LIN {X 0.105,Y -185.624,Z 1374.736,A 0.000,B 0.000,C 90.000,E1 132.528} C_DIS
LIN {X -0.109,Y -190.219,Z 1374.723,A 0.000,B 0.000,C 90.000,E1 130.092} C_DIS
LIN {X 0.050,Y -197.547,Z 1374.700,A 0.000,B 0.000,C 90.000,E1 125.931} C_DIS
LIN {X -0.069,Y -199.265,Z 1374.695,A 0.000,B 0.000,C 90.000,E1 125.105} C_DIS
LIN {X -0.160,Y -309.469,Z 1374.695,A 0.000,B 0.000,C 90.000,E1 125.105} C_DIS
LIN {X -0.107,Y -315.167,Z 1374.694,A 0.000,B 0.000,C 90.000,E1 124.898} C_DIS
LIN {X 0.002,Y -317.632,Z 1374.693,A 0.000,B 0.000,C 90.000,E1 124.692} C_DIS
LIN {X -0.039,Y -320.942,Z 1374.691,A 0.000,B 0.000,C 90.000,E1 124.326} C_DIS
LIN {X 0.118,Y -322.871,Z 1374.689,A 0.000,B 0.000,C 90.000,E1 123.992} C_DIS
LIN {X 0.008,Y -324.375,Z 1374.687,A 0.000,B 0.000,C 90.000,E1 123.706} C_DIS
LIN {X -0.049,Y -330.062,Z 1374.678,A 0.000,B 0.000,C 90.000,E1 122.133} C_DIS
LIN {X -0.113,Y -341.033,Z 1374.663,A 0.000,B 0.000,C 90.000,E1 119.333} C_DIS
LIN {X -0.049,Y -353.383,Z 1374.648,A 0.000,B 0.000,C 90.000,E1 116.565} C_DIS
LIN {X 0.221,Y -367.224,Z 1374.633,A 0.000,B 0.000,C 90.000,E1 113.823} C_DIS
LIN {X -0.172,Y -380.873,Z 1374.620,A 0.000,B 0.000,C 90.000,E1 111.535} C_DIS
LIN {X -0.009,Y -395.888,Z 1374.607,A 0.000,B 0.000,C 90.000,E1 109.214} C_DIS
LIN {X -0.103,Y -412.375,Z 1374.594,A 0.000,B 0.000,C 90.000,E1 106.985} C_DIS
LIN {X 0.086,Y -430.447,Z 1374.582,A 0.000,B 0.000,C 90.000,E1 104.773} C_DIS
LIN {X 0.229,Y -450.044,Z 1374.570,A 0.000,B 0.000,C 90.000,E1 102.647} C_DIS
LIN {X 0.127,Y -470.327,Z 1374.560,A 0.000,B 0.000,C 90.000,E1 100.715} C_DIS
LIN {X -0.144,Y -483.065,Z 1374.553,A 0.000,B 0.000,C 90.000,E1 99.613} C_DIS
LIN {X -0.024,Y -484.891,Z 1374.552,A 0.000,B 0.000,C 90.000,E1 99.378} C_DIS
LIN {X -0.216,Y -486.450,Z 1374.551,A 0.000,B 0.000,C 90.000,E1 99.151} C_DIS
LIN {X 0.153,Y -487.615,Z 1374.549,A 0.000,B 0.000,C 90.000,E1 98.859} C_DIS
LIN {X -0.131,Y -489.012,Z 1374.547,A 0.000,B 0.000,C 90.000,E1 98.398} C_DIS
LIN {X 0.145,Y -489.364,Z 1374.544,A 0.000,B 0.000,C 90.000,E1 97.871} C_DIS
LIN {X -0.125,Y -488.733,Z 1374.541,A 0.000,B 0.000,C 90.000,E1 97.409} C_DIS
LIN {X 0.092,Y -487.015,Z 1374.538,A 0.000,B 0.000,C 90.000,E1 96.891} C_DIS
LIN {X -0.071,Y -485.649,Z 1374.537,A 0.000,B 0.000,C 90.000,E1 96.663} C_DIS
LIN {X -0.175,Y -473.603,Z 1374.527,A 0.000,B 0.000,C 90.000,E1 94.935} C_DIS
LIN {X 0.126,Y -463.887,Z 1374.519,A 0.000,B 0.000,C 90.000,E1 93.383} C_DIS
LIN {X 0.197,Y -447.231,Z 1374.505,A 0.000,B 0.000,C 90.000,E1 90.802} C_DIS
LIN {X -0.052,Y -430.569,Z 1374.489,A 0.000,B 0.000,C 90.000,E1 87.936} C_DIS
LIN {X 0.031,Y -420.205,Z 1374.478,A 0.000,B 0.000,C 90.000,E1 86.045} C_DIS
LIN {X -0.127,Y -411.195,Z 1374.469,A 0.000,B 0.000,C 90.000,E1 84.432} C_DIS
LIN {X -0.029,Y -402.061,Z 1374.460,A 0.000,B 0.000,C 90.000,E1 82.761} C_DIS
LIN {X -0.049,Y -392.775,Z 1374.450,A 0.000,B 0.000,C 90.000,E1 81.084} C_DIS
LIN {X -0.172,Y -383.322,Z 1374.441,A 0.000,B 0.000,C 90.000,E1 79.398} C_DIS
LIN {X -0.019,Y -373.672,Z 1374.431,A 0.000,B 0.000,C 90.000,E1 77.645} C_DIS
LIN {X 0.006,Y -362.297,Z 1374.420,A 0.000,B 0.000,C 90.000,E1 75.589} C_DIS
LIN {X 0.034,Y -352.345,Z 1374.410,A 0.000,B 0.000,C 90.000,E1 73.795} C_DIS
LIN {X -0.097,Y -340.586,Z 1374.398,A 0.000,B 0.000,C 90.000,E1 71.692} C_DIS
LIN {X -0.079,Y -327.270,Z 1374.384,A 0.000,B 0.000,C 90.000,E1 69.209} C_DIS
LIN {X 0.144,Y -309.803,Z 1374.365,A 0.000,B 0.000,C 90.000,E1 65.665} C_DIS
LIN {X 0.004,Y -298.357,Z 1374.350,A 0.000,B 0.000,C 90.000,E1 63.076} C_DIS
LIN {X -0.008,Y -288.146,Z 1374.336,A 0.000,B 0.000,C 90.000,E1 60.411} C_DIS
LIN {X -0.037,Y -280.120,Z 1374.322,A 0.000,B 0.000,C 90.000,E1 58.043} C_DIS
LIN {X -0.094,Y -269.766,Z 1374.303,A 0.000,B 0.000,C 90.000,E1 54.609} C_DIS
LIN {X 0.025,Y -261.942,Z 1374.288,A 0.000,B 0.000,C 90.000,E1 51.778} C_DIS
LIN {X -0.109,Y -252.668,Z 1374.268,A 0.000,B 0.000,C 90.000,E1 48.243} C_DIS
LIN {X -0.031,Y -243.965,Z 1374.248,A 0.000,B 0.000,C 90.000,E1 44.595} C_DIS
LIN {X -0.046,Y -236.060,Z 1374.227,A 0.000,B 0.000,C 90.000,E1 40.906} C_DIS
LIN {X -0.053,Y -229.071,Z 1374.206,A 0.000,B 0.000,C 90.000,E1 37.156} C_DIS
LIN {X -0.129,Y -223.036,Z 1374.185,A 0.000,B 0.000,C 90.000,E1 33.372} C_DIS
LIN {X -0.004,Y -217.876,Z 1374.164,A 0.000,B 0.000,C 90.000,E1 29.489} C_DIS
LIN {X -0.036,Y -213.025,Z 1374.138,A 0.000,B 0.000,C 90.000,E1 24.823} C_DIS
LIN {X -0.067,Y -209.079,Z 1374.107,A 0.000,B 0.000,C 90.000,E1 19.322} C_DIS
LIN {X -0.103,Y -206.893,Z 1374.085,A 0.000,B 0.000,C 90.000,E1 15.371} C_DIS
LIN {X -0.057,Y -205.266,Z 1374.068,A 0.000,B 0.000,C 90.000,E1 12.175} C_DIS
LIN {X 0.007,Y -203.473,Z 1374.045,A 0.000,B 0.000,C 90.000,E1 8.163} C_DIS
LIN {X 0.081,Y -202.199,Z 1374.028,A 0.000,B 0.000,C 90.000,E1 4.935} C_DIS
LIN {X 0.072,Y -200.811,Z 1374.005,A 0.000,B 0.000,C 90.000,E1 0.917} C_DIS
LIN {X -0.095,Y -199.758,Z 1373.979,A 0.000,B 0.000,C 90.000,E1 356.331} C_DIS
LIN {X -0.074,Y -199.675,Z 1373.944,A 0.000,B 0.000,C 90.000,E1 349.859} C_DIS
LIN {X -0.085,Y -201.962,Z 1373.903,A 0.000,B 0.000,C 90.000,E1 342.598} C_DIS
LIN {X 0.056,Y -205.049,Z 1373.876,A 0.000,B 0.000,C 90.000,E1 337.741} C_DIS
LIN {X 0.008,Y -208.842,Z 1373.854,A 0.000,B 0.000,C 90.000,E1 333.768} C_DIS
LIN {X 0.092,Y -213.731,Z 1373.832,A 0.000,B 0.000,C 90.000,E1 329.793} C_DIS
LIN {X 0.106,Y -219.917,Z 1373.811,A 0.000,B 0.000,C 90.000,E1 325.881} C_DIS
LIN {X -0.049,Y -227.282,Z 1373.789,A 0.000,B 0.000,C 90.000,E1 322.065} C_DIS
LIN {X -0.010,Y -234.219,Z 1373.772,A 0.000,B 0.000,C 90.000,E1 319.013} C_DIS
LIN {X -0.023,Y -242.957,Z 1373.754,A 0.000,B 0.000,C 90.000,E1 315.648} C_DIS
LIN {X -0.114,Y -252.763,Z 1373.735,A 0.000,B 0.000,C 90.000,E1 312.366} C_DIS
LIN {X 0.056,Y -261.458,Z 1373.721,A 0.000,B 0.000,C 90.000,E1 309.806} C_DIS
LIN {X -0.038,Y -272.553,Z 1373.705,A 0.000,B 0.000,C 90.000,E1 306.996} C_DIS
LIN {X 0.034,Y -281.723,Z 1373.694,A 0.000,B 0.000,C 90.000,E1 304.898} C_DIS
LIN {X -0.087,Y -290.252,Z 1373.684,A 0.000,B 0.000,C 90.000,E1 303.214} C_DIS
LIN {X -0.145,Y -299.719,Z 1373.675,A 0.000,B 0.000,C 90.000,E1 301.544} C_DIS
LIN {X -0.081,Y -308.351,Z 1373.668,A 0.000,B 0.000,C 90.000,E1 300.207} C_DIS
LIN {X 0.118,Y -317.891,Z 1373.661,A 0.000,B 0.000,C 90.000,E1 298.871} C_DIS
LIN {X -0.069,Y -341.252,Z 1373.645,A 0.000,B 0.000,C 90.000,E1 296.155} C_DIS
LIN {X 0.073,Y -357.170,Z 1373.635,A 0.000,B 0.000,C 90.000,E1 294.387} C_DIS
LIN {X 0.007,Y -370.314,Z 1373.628,A 0.000,B 0.000,C 90.000,E1 292.950} C_DIS
LIN {X -0.170,Y -383.139,Z 1373.620,A 0.000,B 0.000,C 90.000,E1 291.535} C_DIS
LIN {X 0.068,Y -395.535,Z 1373.612,A 0.000,B 0.000,C 90.000,E1 290.066} C_DIS
LIN {X -0.132,Y -415.163,Z 1373.599,A 0.000,B 0.000,C 90.000,E1 287.873} C_DIS
LIN {X -0.057,Y -422.593,Z 1373.595,A 0.000,B 0.000,C 90.000,E1 287.040} C_DIS
LIN {X 0.097,Y -429.432,Z 1373.590,A 0.000,B 0.000,C 90.000,E1 286.205} C_DIS
LIN {X -0.108,Y -435.752,Z 1373.586,A 0.000,B 0.000,C 90.000,E1 285.426} C_DIS
LIN {X 0.167,Y -441.277,Z 1373.581,A 0.000,B 0.000,C 90.000,E1 284.592} C_DIS
LIN {X -0.050,Y -446.081,Z 1373.577,A 0.000,B 0.000,C 90.000,E1 283.828} C_DIS
LIN {X -0.220,Y -450.004,Z 1373.572,A 0.000,B 0.000,C 90.000,E1 283.063} C_DIS
LIN {X 0.082,Y -453.203,Z 1373.568,A 0.000,B 0.000,C 90.000,E1 282.243} C_DIS
LIN {X 0.156,Y -454.826,Z 1373.565,A 0.000,B 0.000,C 90.000,E1 281.715} C_DIS
LIN {X -0.213,Y -456.108,Z 1373.562,A 0.000,B 0.000,C 90.000,E1 281.243} C_DIS
LIN {X -0.128,Y -456.942,Z 1373.559,A 0.000,B 0.000,C 90.000,E1 280.715} C_DIS
LIN {X -0.118,Y -457.349,Z 1373.557,A 0.000,B 0.000,C 90.000,E1 280.197} C_DIS
LIN {X -0.022,Y -457.353,Z 1373.554,A 0.000,B 0.000,C 90.000,E1 279.670} C_DIS
LIN {X 0.000,Y -456.869,Z 1373.551,A 0.000,B 0.000,C 90.000,E1 279.151} C_DIS
LIN {X 0.094,Y -455.930,Z 1373.548,A 0.000,B 0.000,C 90.000,E1 278.624} C_DIS
LIN {X 0.115,Y -454.459,Z 1373.545,A 0.000,B 0.000,C 90.000,E1 278.106} C_DIS
LIN {X 0.133,Y -452.478,Z 1373.542,A 0.000,B 0.000,C 90.000,E1 277.587} C_DIS
LIN {X 0.144,Y -449.961,Z 1373.539,A 0.000,B 0.000,C 90.000,E1 277.068} C_DIS
LIN {X 0.137,Y -446.826,Z 1373.536,A 0.000,B 0.000,C 90.000,E1 276.549} C_DIS
LIN {X 0.115,Y -442.922,Z 1373.534,A 0.000,B 0.000,C 90.000,E1 276.030} C_DIS
LIN {X 0.072,Y -438.005,Z 1373.531,A 0.000,B 0.000,C 90.000,E1 275.511} C_DIS
LIN {X -0.117,Y -435.182,Z 1373.529,A 0.000,B 0.000,C 90.000,E1 275.277} C_DIS
LIN {X 0.169,Y -429.024,Z 1373.527,A 0.000,B 0.000,C 90.000,E1 274.759} C_DIS
LIN {X 0.043,Y -422.617,Z 1373.524,A 0.000,B 0.000,C 90.000,E1 274.359} C_DIS
LIN {X -0.085,Y -416.040,Z 1373.522,A 0.000,B 0.000,C 90.000,E1 274.012} C_DIS
LIN {X 0.069,Y -409.422,Z 1373.520,A 0.000,B 0.000,C 90.000,E1 273.669} C_DIS
LIN {X -0.047,Y -399.427,Z 1373.518,A 0.000,B 0.000,C 90.000,E1 273.269} C_DIS
LIN {X -0.068,Y -389.737,Z 1373.516,A 0.000,B 0.000,C 90.000,E1 272.922} C_DIS
LIN {X 0.037,Y -382.812,Z 1373.515,A 0.000,B 0.000,C 90.000,E1 272.694} C_DIS
LIN {X -0.053,Y -375.514,Z 1373.514,A 0.000,B 0.000,C 90.000,E1 272.522} C_DIS
LIN {X 0.066,Y -367.884,Z 1373.513,A 0.000,B 0.000,C 90.000,E1 272.350} C_DIS
LIN {X -0.002,Y -356.175,Z 1373.512,A 0.000,B 0.000,C 90.000,E1 272.178} C_DIS
LIN {X 0.066,Y -346.221,Z 1373.511,A 0.000,B 0.000,C 90.000,E1 272.064} C_DIS
LIN {X -0.072,Y -330.914,Z 1373.511,A 0.000,B 0.000,C 90.000,E1 272.007} C_DIS
LIN {X -0.116,Y -327.857,Z 1373.511,A 0.000,B 0.000,C 90.000,E1 272.007} C_DIS
LIN {X -0.089,Y -181.265,Z 1373.511,A 0.000,B 0.000,C 90.000,E1 272.007} C_DIS
LIN {X 0.058,Y -181.581,Z 1373.501,A 0.000,B 0.000,C 90.000,E1 270.229} C_DIS
LIN {X 0.046,Y -180.895,Z 1373.473,A 0.000,B 0.000,C 90.000,E1 265.179} C_DIS
LIN {X 0.053,Y -179.837,Z 1373.459,A 0.000,B 0.000,C 90.000,E1 262.648} C_DIS
LIN {X -0.068,Y -179.024,Z 1373.445,A 0.000,B 0.000,C 90.000,E1 260.151} C_DIS
LIN {X -0.006,Y -178.664,Z 1373.440,A 0.000,B 0.000,C 90.000,E1 259.285} C_DIS
LIN {X -0.070,Y -175.715,Z 1373.412,A 0.000,B 0.000,C 90.000,E1 254.212} C_DIS
LIN {X -0.053,Y -172.430,Z 1373.388,A 0.000,B 0.000,C 90.000,E1 249.934} C_DIS
LIN {X -0.033,Y -171.258,Z 1373.379,A 0.000,B 0.000,C 90.000,E1 248.209} C_DIS
LIN {X -0.050,Y -167.529,Z 1373.355,A 0.000,B 0.000,C 90.000,E1 243.896} C_DIS
LIN {X 0.033,Y -166.925,Z 1373.350,A 0.000,B 0.000,C 90.000,E1 242.999} C_DIS
LIN {X -0.046,Y -162.921,Z 1373.326,A 0.000,B 0.000,C 90.000,E1 238.663} C_DIS
LIN {X -0.068,Y -161.594,Z 1373.316,A 0.000,B 0.000,C 90.000,E1 236.914} C_DIS
LIN {X 0.058,Y -158.336,Z 1373.296,A 0.000,B 0.000,C 90.000,E1 233.336} C_DIS
LIN {X -0.081,Y -155.638,Z 1373.277,A 0.000,B 0.000,C 90.000,E1 229.828} C_DIS
LIN {X -0.026,Y -151.911,Z 1373.252,A 0.000,B 0.000,C 90.000,E1 225.324} C_DIS
LIN {X -0.012,Y -150.145,Z 1373.237,A 0.000,B 0.000,C 90.000,E1 222.609} C_DIS
LIN {X 0.026,Y -146.929,Z 1373.211,A 0.000,B 0.000,C 90.000,E1 218.051} C_DIS
LIN {X 0.017,Y -145.517,Z 1373.196,A 0.000,B 0.000,C 90.000,E1 215.311} C_DIS
LIN {X 0.011,Y -142.917,Z 1373.171,A 0.000,B 0.000,C 90.000,E1 210.718} C_DIS
LIN {X 0.064,Y -141.540,Z 1373.150,A 0.000,B 0.000,C 90.000,E1 207.001} C_DIS
LIN {X -0.024,Y -139.401,Z 1373.114,A 0.000,B 0.000,C 90.000,E1 200.536} C_DIS
LIN {X -0.019,Y -139.118,Z 1373.104,A 0.000,B 0.000,C 90.000,E1 198.671} C_DIS
LIN {X 0.013,Y -138.352,Z 1373.057,A 0.000,B 0.000,C 90.000,E1 190.254} C_DIS
LIN {X 0.003,Y -139.505,Z 1373.005,A 0.000,B 0.000,C 90.000,E1 180.917} C_DIS
LIN {X -0.056,Y -141.138,Z 1372.974,A 0.000,B 0.000,C 90.000,E1 175.355} C_DIS
LIN {X 0.038,Y -142.518,Z 1372.959,A 0.000,B 0.000,C 90.000,E1 172.534} C_DIS
LIN {X -0.017,Y -144.780,Z 1372.933,A 0.000,B 0.000,C 90.000,E1 167.937} C_DIS
LIN {X -0.029,Y -147.396,Z 1372.912,A 0.000,B 0.000,C 90.000,E1 164.267} C_DIS
LIN {X 0.002,Y -149.970,Z 1372.892,A 0.000,B 0.000,C 90.000,E1 160.604} C_DIS
LIN {X 0.012,Y -153.292,Z 1372.872,A 0.000,B 0.000,C 90.000,E1 156.975} C_DIS
LIN {X -0.001,Y -154.996,Z 1372.862,A 0.000,B 0.000,C 90.000,E1 155.177} C_DIS
LIN {X 0.012,Y -158.636,Z 1372.842,A 0.000,B 0.000,C 90.000,E1 151.591} C_DIS
LIN {X -0.051,Y -161.910,Z 1372.827,A 0.000,B 0.000,C 90.000,E1 148.948} C_DIS
LIN {X 0.057,Y -166.100,Z 1372.808,A 0.000,B 0.000,C 90.000,E1 145.388} C_DIS
LIN {X 0.055,Y -171.109,Z 1372.788,A 0.000,B 0.000,C 90.000,E1 141.904} C_DIS
LIN {X -0.026,Y -175.985,Z 1372.769,A 0.000,B 0.000,C 90.000,E1 138.485} C_DIS
LIN {X 0.088,Y -180.232,Z 1372.755,A 0.000,B 0.000,C 90.000,E1 135.891} C_DIS
LIN {X 0.062,Y -185.646,Z 1372.736,A 0.000,B 0.000,C 90.000,E1 132.528} C_DIS
LIN {X 0.115,Y -190.244,Z 1372.723,A 0.000,B 0.000,C 90.000,E1 130.011} C_DIS
LIN {X 0.006,Y -197.572,Z 1372.700,A 0.000,B 0.000,C 90.000,E1 125.931} C_DIS
LIN {X -0.047,Y -199.252,Z 1372.695,A 0.000,B 0.000,C 90.000,E1 125.105} C_DIS
LIN {X -0.125,Y -309.511,Z 1372.695,A 0.000,B 0.000,C 90.000,E1 125.105} C_DIS
LIN {X 0.151,Y -311.252,Z 1372.695,A 0.000,B 0.000,C 90.000,E1 125.025} C_DIS
LIN {X -0.178,Y -315.434,Z 1372.694,A 0.000,B 0.000,C 90.000,E1 124.898} C_DIS
LIN {X -0.069,Y -317.806,Z 1372.693,A 0.000,B 0.000,C 90.000,E1 124.692} C_DIS
LIN {X -0.111,Y -321.038,Z 1372.691,A 0.000,B 0.000,C 90.000,E1 124.326} C_DIS
LIN {X 0.018,Y -322.962,Z 1372.689,A 0.000,B 0.000,C 90.000,E1 123.992} C_DIS
LIN {X -0.122,Y -324.459,Z 1372.687,A 0.000,B 0.000,C 90.000,E1 123.706} C_DIS
LIN {X -0.065,Y -338.549,Z 1372.666,A 0.000,B 0.000,C 90.000,E1 119.922} C_DIS
LIN {X 0.086,Y -350.594,Z 1372.651,A 0.000,B 0.000,C 90.000,E1 117.129} C_DIS
LIN {X -0.208,Y -364.107,Z 1372.636,A 0.000,B 0.000,C 90.000,E1 114.463} C_DIS
LIN {X -0.051,Y -377.441,Z 1372.623,A 0.000,B 0.000,C 90.000,E1 112.078} C_DIS
LIN {X 0.021,Y -392.117,Z 1372.610,A 0.000,B 0.000,C 90.000,E1 109.758} C_DIS
LIN {X -0.043,Y -408.239,Z 1372.597,A 0.000,B 0.000,C 90.000,E1 107.511} C_DIS
LIN {X 0.036,Y -425.918,Z 1372.585,A 0.000,B 0.000,C 90.000,E1 105.300} C_DIS
LIN {X -0.042,Y -445.220,Z 1372.573,A 0.000,B 0.000,C 90.000,E1 103.175} C_DIS
LIN {X -0.025,Y -465.369,Z 1372.562,A 0.000,B 0.000,C 90.000,E1 101.186} C_DIS
LIN {X 0.067,Y -480.831,Z 1372.554,A 0.000,B 0.000,C 90.000,E1 99.792} C_DIS
LIN {X 0.191,Y -483.168,Z 1372.553,A 0.000,B 0.000,C 90.000,E1 99.557} C_DIS
LIN {X -0.165,Y -484.936,Z 1372.552,A 0.000,B 0.000,C 90.000,E1 99.378} C_DIS
LIN {X 0.124,Y -486.450,Z 1372.551,A 0.000,B 0.000,C 90.000,E1 99.095} C_DIS
LIN {X 0.012,Y -487.579,Z 1372.549,A 0.000,B 0.000,C 90.000,E1 98.859} C_DIS
LIN {X 0.212,Y -488.916,Z 1372.547,A 0.000,B 0.000,C 90.000,E1 98.341} C_DIS
LIN {X 0.004,Y -489.218,Z 1372.544,A 0.000,B 0.000,C 90.000,E1 97.871} C_DIS
LIN {X 0.217,Y -488.536,Z 1372.541,A 0.000,B 0.000,C 90.000,E1 97.352} C_DIS
LIN {X -0.050,Y -486.756,Z 1372.538,A 0.000,B 0.000,C 90.000,E1 96.891} C_DIS
LIN {X -0.213,Y -485.350,Z 1372.537,A 0.000,B 0.000,C 90.000,E1 96.663} C_DIS
LIN {X 0.151,Y -473.261,Z 1372.527,A 0.000,B 0.000,C 90.000,E1 94.878} C_DIS
LIN {X -0.022,Y -463.534,Z 1372.519,A 0.000,B 0.000,C 90.000,E1 93.383} C_DIS
LIN {X 0.044,Y -446.887,Z 1372.505,A 0.000,B 0.000,C 90.000,E1 90.802} C_DIS
LIN {X -0.209,Y -430.250,Z 1372.488,A 0.000,B 0.000,C 90.000,E1 87.936} C_DIS
LIN {X -0.129,Y -419.902,Z 1372.478,A 0.000,B 0.000,C 90.000,E1 86.045} C_DIS
LIN {X 0.192,Y -409.407,Z 1372.467,A 0.000,B 0.000,C 90.000,E1 84.090} C_DIS
LIN {X -0.103,Y -400.252,Z 1372.458,A 0.000,B 0.000,C 90.000,E1 82.470} C_DIS
LIN {X -0.150,Y -390.950,Z 1372.449,A 0.000,B 0.000,C 90.000,E1 80.792} C_DIS
LIN {X 0.107,Y -379.869,Z 1372.438,A 0.000,B 0.000,C 90.000,E1 78.757} C_DIS
LIN {X -0.097,Y -368.549,Z 1372.426,A 0.000,B 0.000,C 90.000,E1 76.756} C_DIS
LIN {X -0.132,Y -358.725,Z 1372.417,A 0.000,B 0.000,C 90.000,E1 74.991} C_DIS
LIN {X 0.174,Y -348.741,Z 1372.406,A 0.000,B 0.000,C 90.000,E1 73.142} C_DIS
LIN {X -0.040,Y -336.998,Z 1372.395,A 0.000,B 0.000,C 90.000,E1 71.040} C_DIS
LIN {X -0.008,Y -323.745,Z 1372.381,A 0.000,B 0.000,C 90.000,E1 68.539} C_DIS
LIN {X -0.020,Y -309.564,Z 1372.365,A 0.000,B 0.000,C 90.000,E1 65.665} C_DIS
LIN {X -0.024,Y -298.147,Z 1372.350,A 0.000,B 0.000,C 90.000,E1 63.050} C_DIS
LIN {X -0.040,Y -286.763,Z 1372.334,A 0.000,B 0.000,C 90.000,E1 60.049} C_DIS
LIN {X 0.016,Y -275.761,Z 1372.315,A 0.000,B 0.000,C 90.000,E1 56.628} C_DIS
LIN {X 0.128,Y -265.744,Z 1372.295,A 0.000,B 0.000,C 90.000,E1 53.130} C_DIS
LIN {X -0.020,Y -256.269,Z 1372.276,A 0.000,B 0.000,C 90.000,E1 49.622} C_DIS
LIN {X 0.173,Y -247.360,Z 1372.256,A 0.000,B 0.000,C 90.000,E1 45.972} C_DIS
LIN {X -0.092,Y -239.161,Z 1372.235,A 0.000,B 0.000,C 90.000,E1 42.366} C_DIS
LIN {X -0.033,Y -231.820,Z 1372.214,A 0.000,B 0.000,C 90.000,E1 38.624} C_DIS
LIN {X 0.055,Y -225.418,Z 1372.193,A 0.000,B 0.000,C 90.000,E1 34.818} C_DIS
LIN {X -0.013,Y -219.937,Z 1372.172,A 0.000,B 0.000,C 90.000,E1 31.003} C_DIS
LIN {X -0.017,Y -215.399,Z 1372.151,A 0.000,B 0.000,C 90.000,E1 27.129} C_DIS
LIN {X -0.126,Y -211.288,Z 1372.125,A 0.000,B 0.000,C 90.000,E1 22.461} C_DIS
LIN {X -0.022,Y -208.795,Z 1372.103,A 0.000,B 0.000,C 90.000,E1 18.489} C_DIS
LIN {X -0.064,Y -206.647,Z 1372.081,A 0.000,B 0.000,C 90.000,E1 14.537} C_DIS
LIN {X -0.114,Y -205.032,Z 1372.063,A 0.000,B 0.000,C 90.000,E1 11.366} C_DIS
LIN {X -0.052,Y -203.276,Z 1372.041,A 0.000,B 0.000,C 90.000,E1 7.352} C_DIS
LIN {X -0.003,Y -202.025,Z 1372.023,A 0.000,B 0.000,C 90.000,E1 4.131} C_DIS
LIN {X 0.000,Y -200.675,Z 1372.000,A 0.000,B 0.000,C 90.000,E1 360.000} C_DIS
LIN {X 0.082,Y -199.689,Z 1371.970,A 0.000,B 0.000,C 90.000,E1 354.666} C_DIS
LIN {X -0.016,Y -200.077,Z 1371.935,A 0.000,B 0.000,C 90.000,E1 348.229} C_DIS
LIN {X 0.037,Y -202.542,Z 1371.899,A 0.000,B 0.000,C 90.000,E1 341.764} C_DIS
LIN {X -0.035,Y -205.889,Z 1371.872,A 0.000,B 0.000,C 90.000,E1 336.975} C_DIS
LIN {X -0.051,Y -209.898,Z 1371.850,A 0.000,B 0.000,C 90.000,E1 332.999} C_DIS
LIN {X -0.125,Y -215.041,Z 1371.828,A 0.000,B 0.000,C 90.000,E1 329.076} C_DIS
LIN {X 0.038,Y -221.503,Z 1371.806,A 0.000,B 0.000,C 90.000,E1 325.135} C_DIS
LIN {X 0.003,Y -227.470,Z 1371.789,A 0.000,B 0.000,C 90.000,E1 322.065} C_DIS
LIN {X 0.048,Y -234.398,Z 1371.772,A 0.000,B 0.000,C 90.000,E1 319.013} C_DIS
LIN {X 0.042,Y -243.099,Z 1371.754,A 0.000,B 0.000,C 90.000,E1 315.648} C_DIS
LIN {X -0.042,Y -252.882,Z 1371.735,A 0.000,B 0.000,C 90.000,E1 312.366} C_DIS
LIN {X -0.068,Y -261.572,Z 1371.721,A 0.000,B 0.000,C 90.000,E1 309.850} C_DIS
LIN {X -0.036,Y -271.198,Z 1371.708,A 0.000,B 0.000,C 90.000,E1 307.363} C_DIS
LIN {X 0.121,Y -281.843,Z 1371.694,A 0.000,B 0.000,C 90.000,E1 304.898} C_DIS
LIN {X 0.005,Y -290.386,Z 1371.685,A 0.000,B 0.000,C 90.000,E1 303.214} C_DIS
LIN {X -0.052,Y -297.857,Z 1371.677,A 0.000,B 0.000,C 90.000,E1 301.878} C_DIS
LIN {X -0.027,Y -304.002,Z 1371.672,A 0.000,B 0.000,C 90.000,E1 300.875} C_DIS
LIN {X 0.096,Y -313.091,Z 1371.664,A 0.000,B 0.000,C 90.000,E1 299.539} C_DIS
LIN {X -0.034,Y -323.051,Z 1371.657,A 0.000,B 0.000,C 90.000,E1 298.281} C_DIS
LIN {X -0.070,Y -344.190,Z 1371.644,A 0.000,B 0.000,C 90.000,E1 295.848} C_DIS
LIN {X -0.108,Y -357.584,Z 1371.635,A 0.000,B 0.000,C 90.000,E1 294.387} C_DIS
LIN {X -0.144,Y -370.669,Z 1371.627,A 0.000,B 0.000,C 90.000,E1 292.950} C_DIS
LIN {X 0.171,Y -383.441,Z 1371.619,A 0.000,B 0.000,C 90.000,E1 291.461} C_DIS
LIN {X -0.041,Y -395.776,Z 1371.611,A 0.000,B 0.000,C 90.000,E1 290.066} C_DIS
LIN {X 0.041,Y -415.525,Z 1371.599,A 0.000,B 0.000,C 90.000,E1 287.819} C_DIS
LIN {X 0.122,Y -422.909,Z 1371.594,A 0.000,B 0.000,C 90.000,E1 286.985} C_DIS
LIN {X -0.131,Y -429.736,Z 1371.590,A 0.000,B 0.000,C 90.000,E1 286.205} C_DIS
LIN {X -0.092,Y -434.032,Z 1371.587,A 0.000,B 0.000,C 90.000,E1 285.662} C_DIS
LIN {X 0.160,Y -439.810,Z 1371.583,A 0.000,B 0.000,C 90.000,E1 284.828} C_DIS
LIN {X -0.065,Y -444.862,Z 1371.578,A 0.000,B 0.000,C 90.000,E1 284.064} C_DIS
LIN {X 0.186,Y -449.066,Z 1371.574,A 0.000,B 0.000,C 90.000,E1 283.244} C_DIS
LIN {X 0.046,Y -452.488,Z 1371.569,A 0.000,B 0.000,C 90.000,E1 282.479} C_DIS
LIN {X -0.144,Y -453.489,Z 1371.568,A 0.000,B 0.000,C 90.000,E1 282.243} C_DIS
LIN {X -0.070,Y -455.105,Z 1371.565,A 0.000,B 0.000,C 90.000,E1 281.715} C_DIS
LIN {X 0.010,Y -456.385,Z 1371.562,A 0.000,B 0.000,C 90.000,E1 281.186} C_DIS
LIN {X 0.098,Y -457.229,Z 1371.559,A 0.000,B 0.000,C 90.000,E1 280.658} C_DIS
LIN {X 0.110,Y -457.630,Z 1371.556,A 0.000,B 0.000,C 90.000,E1 280.141} C_DIS
LIN {X 0.208,Y -457.616,Z 1371.554,A 0.000,B 0.000,C 90.000,E1 279.613} C_DIS
LIN {X -0.219,Y -457.147,Z 1371.551,A 0.000,B 0.000,C 90.000,E1 279.151} C_DIS
LIN {X -0.122,Y -456.161,Z 1371.548,A 0.000,B 0.000,C 90.000,E1 278.624} C_DIS
LIN {X -0.099,Y -454.686,Z 1371.545,A 0.000,B 0.000,C 90.000,E1 278.106} C_DIS
LIN {X -0.079,Y -452.731,Z 1371.542,A 0.000,B 0.000,C 90.000,E1 277.587} C_DIS
LIN {X -0.065,Y -450.174,Z 1371.539,A 0.000,B 0.000,C 90.000,E1 277.068} C_DIS
LIN {X -0.069,Y -447.038,Z 1371.536,A 0.000,B 0.000,C 90.000,E1 276.549} C_DIS
LIN {X -0.089,Y -443.104,Z 1371.533,A 0.000,B 0.000,C 90.000,E1 276.030} C_DIS
LIN {X -0.129,Y -438.295,Z 1371.531,A 0.000,B 0.000,C 90.000,E1 275.511} C_DIS
LIN {X -0.126,Y -432.278,Z 1371.528,A 0.000,B 0.000,C 90.000,E1 274.992} C_DIS
LIN {X -0.006,Y -426.017,Z 1371.525,A 0.000,B 0.000,C 90.000,E1 274.531} C_DIS
LIN {X 0.074,Y -419.486,Z 1371.523,A 0.000,B 0.000,C 90.000,E1 274.131} C_DIS
LIN {X 0.181,Y -413.145,Z 1371.521,A 0.000,B 0.000,C 90.000,E1 273.784} C_DIS
LIN {X -0.067,Y -403.447,Z 1371.519,A 0.000,B 0.000,C 90.000,E1 273.383} C_DIS
LIN {X 0.121,Y -393.506,Z 1371.517,A 0.000,B 0.000,C 90.000,E1 272.980} C_DIS
LIN {X -0.149,Y -383.221,Z 1371.515,A 0.000,B 0.000,C 90.000,E1 272.694} C_DIS
LIN {X 0.147,Y -375.886,Z 1371.514,A 0.000,B 0.000,C 90.000,E1 272.465} C_DIS
LIN {X -0.102,Y -368.080,Z 1371.513,A 0.000,B 0.000,C 90.000,E1 272.350} C_DIS
LIN {X -0.126,Y -356.297,Z 1371.512,A 0.000,B 0.000,C 90.000,E1 272.178} C_DIS
LIN {X -0.049,Y -346.546,Z 1371.511,A 0.000,B 0.000,C 90.000,E1 272.064} C_DIS
LIN {X -0.064,Y -336.433,Z 1371.511,A 0.000,B 0.000,C 90.000,E1 272.007} C_DIS
LIN {X 0.108,Y -326.774,Z 1371.511,A 0.000,B 0.000,C 90.000,E1 271.949} C_DIS
LIN {X 0.036,Y -181.268,Z 1371.511,A 0.000,B 0.000,C 90.000,E1 271.949} C_DIS
LIN {X 0.009,Y -181.580,Z 1371.501,A 0.000,B 0.000,C 90.000,E1 270.229} C_DIS
LIN {X -0.002,Y -180.893,Z 1371.473,A 0.000,B 0.000,C 90.000,E1 265.179} C_DIS
LIN {X 0.075,Y -179.517,Z 1371.454,A 0.000,B 0.000,C 90.000,E1 261.781} C_DIS
LIN {X 0.059,Y -179.020,Z 1371.445,A 0.000,B 0.000,C 90.000,E1 260.095} C_DIS
LIN {X -0.055,Y -178.654,Z 1371.440,A 0.000,B 0.000,C 90.000,E1 259.285} C_DIS
LIN {X 0.051,Y -175.705,Z 1371.412,A 0.000,B 0.000,C 90.000,E1 254.157} C_DIS
LIN {X 0.062,Y -172.420,Z 1371.388,A 0.000,B 0.000,C 90.000,E1 249.880} C_DIS
LIN {X 0.078,Y -171.241,Z 1371.379,A 0.000,B 0.000,C 90.000,E1 248.156} C_DIS
LIN {X 0.053,Y -167.518,Z 1371.355,A 0.000,B 0.000,C 90.000,E1 243.845} C_DIS
LIN {X -0.014,Y -166.914,Z 1371.350,A 0.000,B 0.000,C 90.000,E1 242.999} C_DIS
LIN {X 0.038,Y -162.222,Z 1371.321,A 0.000,B 0.000,C 90.000,E1 237.740} C_DIS
LIN {X -0.043,Y -160.803,Z 1371.311,A 0.000,B 0.000,C 90.000,E1 236.008} C_DIS
LIN {X -0.064,Y -157.590,Z 1371.291,A 0.000,B 0.000,C 90.000,E1 232.477} C_DIS
LIN {X -0.006,Y -155.624,Z 1371.277,A 0.000,B 0.000,C 90.000,E1 229.784} C_DIS
LIN {X -0.071,Y -151.901,Z 1371.252,A 0.000,B 0.000,C 90.000,E1 225.324} C_DIS
LIN {X -0.055,Y -150.131,Z 1371.237,A 0.000,B 0.000,C 90.000,E1 222.609} C_DIS
LIN {X 0.073,Y -146.919,Z 1371.211,A 0.000,B 0.000,C 90.000,E1 218.016} C_DIS
LIN {X -0.026,Y -145.507,Z 1371.196,A 0.000,B 0.000,C 90.000,E1 215.311} C_DIS
LIN {X -0.031,Y -142.910,Z 1371.171,A 0.000,B 0.000,C 90.000,E1 210.718} C_DIS
LIN {X 0.022,Y -141.532,Z 1371.150,A 0.000,B 0.000,C 90.000,E1 207.001} C_DIS
LIN {X 0.065,Y -139.398,Z 1371.114,A 0.000,B 0.000,C 90.000,E1 200.482} C_DIS
LIN {X -0.016,Y -139.112,Z 1371.104,A 0.000,B 0.000,C 90.000,E1 198.652} C_DIS
LIN {X -0.029,Y -138.352,Z 1371.057,A 0.000,B 0.000,C 90.000,E1 190.254} C_DIS
LIN {X -0.039,Y -139.507,Z 1371.005,A 0.000,B 0.000,C 90.000,E1 180.917} C_DIS
LIN {X 0.042,Y -141.146,Z 1370.974,A 0.000,B 0.000,C 90.000,E1 175.298} C_DIS
LIN {X -0.006,Y -142.526,Z 1370.958,A 0.000,B 0.000,C 90.000,E1 172.534} C_DIS
LIN {X -0.060,Y -144.791,Z 1370.933,A 0.000,B 0.000,C 90.000,E1 167.937} C_DIS
LIN {X 0.070,Y -147.408,Z 1370.912,A 0.000,B 0.000,C 90.000,E1 164.212} C_DIS
LIN {X -0.042,Y -149.984,Z 1370.892,A 0.000,B 0.000,C 90.000,E1 160.604} C_DIS
LIN {X -0.033,Y -153.309,Z 1370.872,A 0.000,B 0.000,C 90.000,E1 156.975} C_DIS
LIN {X 0.019,Y -155.011,Z 1370.862,A 0.000,B 0.000,C 90.000,E1 155.153} C_DIS
LIN {X 0.042,Y -158.654,Z 1370.842,A 0.000,B 0.000,C 90.000,E1 151.563} C_DIS
LIN {X -0.013,Y -161.931,Z 1370.827,A 0.000,B 0.000,C 90.000,E1 148.918} C_DIS
LIN {X 0.010,Y -166.122,Z 1370.808,A 0.000,B 0.000,C 90.000,E1 145.388} C_DIS
LIN {X 0.007,Y -171.133,Z 1370.788,A 0.000,B 0.000,C 90.000,E1 141.904} C_DIS
LIN {X -0.074,Y -176.009,Z 1370.769,A 0.000,B 0.000,C 90.000,E1 138.485} C_DIS
LIN {X 0.038,Y -180.260,Z 1370.755,A 0.000,B 0.000,C 90.000,E1 135.891} C_DIS
LIN {X 0.012,Y -185.673,Z 1370.736,A 0.000,B 0.000,C 90.000,E1 132.528} C_DIS
LIN {X 0.064,Y -190.274,Z 1370.722,A 0.000,B 0.000,C 90.000,E1 130.011} C_DIS
LIN {X -0.046,Y -197.602,Z 1370.700,A 0.000,B 0.000,C 90.000,E1 125.931} C_DIS
LIN {X -0.030,Y -199.241,Z 1370.695,A 0.000,B 0.000,C 90.000,E1 125.105} C_DIS
LIN {X -0.082,Y -309.283,Z 1370.695,A 0.000,B 0.000,C 90.000,E1 125.105} C_DIS
LIN {X 0.069,Y -311.968,Z 1370.695,A 0.000,B 0.000,C 90.000,E1 125.025} C_DIS
LIN {X 0.179,Y -315.711,Z 1370.694,A 0.000,B 0.000,C 90.000,E1 124.818} C_DIS
LIN {X -0.152,Y -317.990,Z 1370.693,A 0.000,B 0.000,C 90.000,E1 124.692} C_DIS
LIN {X 0.070,Y -321.147,Z 1370.691,A 0.000,B 0.000,C 90.000,E1 124.278} C_DIS
LIN {X -0.097,Y -323.063,Z 1370.689,A 0.000,B 0.000,C 90.000,E1 123.992} C_DIS
LIN {X 0.004,Y -324.552,Z 1370.687,A 0.000,B 0.000,C 90.000,E1 123.658} C_DIS
LIN {X 0.079,Y -338.629,Z 1370.666,A 0.000,B 0.000,C 90.000,E1 119.873} C_DIS
LIN {X -0.065,Y -350.686,Z 1370.651,A 0.000,B 0.000,C 90.000,E1 117.129} C_DIS
LIN {X 0.120,Y -364.213,Z 1370.636,A 0.000,B 0.000,C 90.000,E1 114.387} C_DIS
LIN {X 0.142,Y -377.560,Z 1370.622,A 0.000,B 0.000,C 90.000,E1 112.025} C_DIS
LIN {X -0.139,Y -392.250,Z 1370.610,A 0.000,B 0.000,C 90.000,E1 109.758} C_DIS
LIN {X 0.184,Y -408.386,Z 1370.597,A 0.000,B 0.000,C 90.000,E1 107.457} C_DIS
LIN {X -0.131,Y -426.083,Z 1370.585,A 0.000,B 0.000,C 90.000,E1 105.300} C_DIS
LIN {X 0.223,Y -445.400,Z 1370.573,A 0.000,B 0.000,C 90.000,E1 103.119} C_DIS
LIN {X -0.187,Y -465.554,Z 1370.562,A 0.000,B 0.000,C 90.000,E1 101.186} C_DIS
LIN {X -0.091,Y -481.020,Z 1370.554,A 0.000,B 0.000,C 90.000,E1 99.792} C_DIS
LIN {X 0.034,Y -483.279,Z 1370.553,A 0.000,B 0.000,C 90.000,E1 99.557} C_DIS
LIN {X 0.157,Y -484.988,Z 1370.552,A 0.000,B 0.000,C 90.000,E1 99.321} C_DIS
LIN {X -0.031,Y -486.454,Z 1370.551,A 0.000,B 0.000,C 90.000,E1 99.095} C_DIS
LIN {X -0.145,Y -487.545,Z 1370.549,A 0.000,B 0.000,C 90.000,E1 98.859} C_DIS
LIN {X 0.055,Y -488.821,Z 1370.546,A 0.000,B 0.000,C 90.000,E1 98.341} C_DIS
LIN {X -0.153,Y -489.070,Z 1370.544,A 0.000,B 0.000,C 90.000,E1 97.871} C_DIS
LIN {X 0.060,Y -488.332,Z 1370.541,A 0.000,B 0.000,C 90.000,E1 97.352} C_DIS
LIN {X -0.208,Y -486.485,Z 1370.538,A 0.000,B 0.000,C 90.000,E1 96.891} C_DIS
LIN {X 0.112,Y -485.034,Z 1370.537,A 0.000,B 0.000,C 90.000,E1 96.606} C_DIS
LIN {X -0.008,Y -472.911,Z 1370.527,A 0.000,B 0.000,C 90.000,E1 94.878} C_DIS
LIN {X -0.184,Y -463.183,Z 1370.519,A 0.000,B 0.000,C 90.000,E1 93.383} C_DIS
LIN {X -0.172,Y -443.375,Z 1370.501,A 0.000,B 0.000,C 90.000,E1 90.286} C_DIS
LIN {X 0.195,Y -428.451,Z 1370.487,A 0.000,B 0.000,C 90.000,E1 87.593} C_DIS
LIN {X -0.168,Y -418.087,Z 1370.476,A 0.000,B 0.000,C 90.000,E1 85.755} C_DIS
LIN {X 0.127,Y -407.602,Z 1370.466,A 0.000,B 0.000,C 90.000,E1 83.799} C_DIS
LIN {X 0.150,Y -398.445,Z 1370.456,A 0.000,B 0.000,C 90.000,E1 82.129} C_DIS
LIN {X 0.120,Y -389.103,Z 1370.447,A 0.000,B 0.000,C 90.000,E1 80.443} C_DIS
LIN {X -0.048,Y -378.005,Z 1370.436,A 0.000,B 0.000,C 90.000,E1 78.465} C_DIS
LIN {X 0.077,Y -366.643,Z 1370.425,A 0.000,B 0.000,C 90.000,E1 76.408} C_DIS
LIN {X 0.090,Y -356.793,Z 1370.415,A 0.000,B 0.000,C 90.000,E1 74.629} C_DIS
LIN {X 0.025,Y -346.803,Z 1370.405,A 0.000,B 0.000,C 90.000,E1 72.834} C_DIS
LIN {X 0.091,Y -335.066,Z 1370.393,A 0.000,B 0.000,C 90.000,E1 70.678} C_DIS
LIN {X 0.188,Y -321.857,Z 1370.379,A 0.000,B 0.000,C 90.000,E1 68.156} C_DIS
LIN {X 0.001,Y -307.825,Z 1370.363,A 0.000,B 0.000,C 90.000,E1 65.305} C_DIS
LIN {X 0.081,Y -296.587,Z 1370.348,A 0.000,B 0.000,C 90.000,E1 62.666} C_DIS
LIN {X 0.012,Y -285.419,Z 1370.332,A 0.000,B 0.000,C 90.000,E1 59.665} C_DIS
LIN {X 0.079,Y -275.649,Z 1370.314,A 0.000,B 0.000,C 90.000,E1 56.580} C_DIS
LIN {X -0.036,Y -265.670,Z 1370.295,A 0.000,B 0.000,C 90.000,E1 53.130} C_DIS
LIN {X -0.015,Y -256.223,Z 1370.276,A 0.000,B 0.000,C 90.000,E1 49.585} C_DIS
LIN {X 0.018,Y -247.334,Z 1370.255,A 0.000,B 0.000,C 90.000,E1 45.972} C_DIS
LIN {X 0.094,Y -239.169,Z 1370.235,A 0.000,B 0.000,C 90.000,E1 42.285} C_DIS
LIN {X -0.035,Y -231.863,Z 1370.214,A 0.000,B 0.000,C 90.000,E1 38.588} C_DIS
LIN {X -0.085,Y -225.489,Z 1370.193,A 0.000,B 0.000,C 90.000,E1 34.818} C_DIS
LIN {X -0.147,Y -220.018,Z 1370.172,A 0.000,B 0.000,C 90.000,E1 31.003} C_DIS
LIN {X 0.046,Y -215.517,Z 1370.151,A 0.000,B 0.000,C 90.000,E1 27.078} C_DIS
LIN {X 0.029,Y -211.454,Z 1370.124,A 0.000,B 0.000,C 90.000,E1 22.386} C_DIS
LIN {X -0.071,Y -208.960,Z 1370.103,A 0.000,B 0.000,C 90.000,E1 18.471} C_DIS
LIN {X 0.027,Y -206.795,Z 1370.080,A 0.000,B 0.000,C 90.000,E1 14.481} C_DIS
LIN {X 0.063,Y -204.808,Z 1370.058,A 0.000,B 0.000,C 90.000,E1 10.489} C_DIS
LIN {X 0.082,Y -203.088,Z 1370.036,A 0.000,B 0.000,C 90.000,E1 6.486} C_DIS
LIN {X -0.092,Y -201.556,Z 1370.014,A 0.000,B 0.000,C 90.000,E1 2.522} C_DIS
LIN {X -0.079,Y -200.124,Z 1369.984,A 0.000,B 0.000,C 90.000,E1 357.135} C_DIS
LIN {X -0.098,Y -199.845,Z 1369.948,A 0.000,B 0.000,C 90.000,E1 350.679} C_DIS
LIN {X 0.039,Y -201.876,Z 1369.908,A 0.000,B 0.000,C 90.000,E1 343.378} C_DIS
LIN {X -0.086,Y -205.399,Z 1369.876,A 0.000,B 0.000,C 90.000,E1 337.794} C_DIS
LIN {X 0.067,Y -209.192,Z 1369.854,A 0.000,B 0.000,C 90.000,E1 333.768} C_DIS
LIN {X -0.129,Y -214.111,Z 1369.832,A 0.000,B 0.000,C 90.000,E1 329.871} C_DIS
LIN {X 0.010,Y -220.320,Z 1369.811,A 0.000,B 0.000,C 90.000,E1 325.928} C_DIS
LIN {X 0.053,Y -227.661,Z 1369.789,A 0.000,B 0.000,C 90.000,E1 322.065} C_DIS
LIN {X 0.104,Y -234.575,Z 1369.772,A 0.000,B 0.000,C 90.000,E1 319.013} C_DIS
LIN {X 0.104,Y -243.246,Z 1369.754,A 0.000,B 0.000,C 90.000,E1 315.648} C_DIS
LIN {X 0.027,Y -253.001,Z 1369.735,A 0.000,B 0.000,C 90.000,E1 312.366} C_DIS
LIN {X 0.007,Y -261.679,Z 1369.721,A 0.000,B 0.000,C 90.000,E1 309.850} C_DIS
LIN {X -0.040,Y -272.749,Z 1369.706,A 0.000,B 0.000,C 90.000,E1 307.030} C_DIS
LIN {X -0.025,Y -281.956,Z 1369.694,A 0.000,B 0.000,C 90.000,E1 304.945} C_DIS
LIN {X -0.064,Y -290.515,Z 1369.685,A 0.000,B 0.000,C 90.000,E1 303.245} C_DIS
LIN {X 0.047,Y -299.955,Z 1369.675,A 0.000,B 0.000,C 90.000,E1 301.544} C_DIS
LIN {X 0.089,Y -306.275,Z 1369.670,A 0.000,B 0.000,C 90.000,E1 300.541} C_DIS
LIN {X -0.032,Y -315.592,Z 1369.662,A 0.000,B 0.000,C 90.000,E1 299.255} C_DIS
LIN {X 0.153,Y -328.331,Z 1369.654,A 0.000,B 0.000,C 90.000,E1 297.641} C_DIS
LIN {X -0.103,Y -347.191,Z 1369.642,A 0.000,B 0.000,C 90.000,E1 295.540} C_DIS
LIN {X -0.055,Y -360.443,Z 1369.634,A 0.000,B 0.000,C 90.000,E1 294.079} C_DIS
LIN {X 0.126,Y -370.886,Z 1369.627,A 0.000,B 0.000,C 90.000,E1 292.898} C_DIS
LIN {X 0.058,Y -383.679,Z 1369.619,A 0.000,B 0.000,C 90.000,E1 291.461} C_DIS
LIN {X -0.146,Y -396.016,Z 1369.611,A 0.000,B 0.000,C 90.000,E1 290.066} C_DIS
LIN {X 0.196,Y -413.269,Z 1369.600,A 0.000,B 0.000,C 90.000,E1 288.055} C_DIS
LIN {X -0.012,Y -423.121,Z 1369.594,A 0.000,B 0.000,C 90.000,E1 286.985} C_DIS
LIN {X 0.149,Y -429.947,Z 1369.590,A 0.000,B 0.000,C 90.000,E1 286.150} C_DIS
LIN {X 0.191,Y -434.243,Z 1369.587,A 0.000,B 0.000,C 90.000,E1 285.607} C_DIS
LIN {X 0.026,Y -440.007,Z 1369.582,A 0.000,B 0.000,C 90.000,E1 284.828} C_DIS
LIN {X -0.199,Y -445.048,Z 1369.578,A 0.000,B 0.000,C 90.000,E1 284.064} C_DIS
LIN {X -0.181,Y -447.982,Z 1369.575,A 0.000,B 0.000,C 90.000,E1 283.536} C_DIS
LIN {X 0.103,Y -451.670,Z 1369.571,A 0.000,B 0.000,C 90.000,E1 282.715} C_DIS
LIN {X 0.168,Y -453.700,Z 1369.568,A 0.000,B 0.000,C 90.000,E1 282.187} C_DIS
LIN {X -0.207,Y -455.380,Z 1369.565,A 0.000,B 0.000,C 90.000,E1 281.715} C_DIS
LIN {X -0.126,Y -456.642,Z 1369.562,A 0.000,B 0.000,C 90.000,E1 281.186} C_DIS
LIN {X -0.037,Y -457.484,Z 1369.559,A 0.000,B 0.000,C 90.000,E1 280.658} C_DIS
LIN {X -0.024,Y -457.921,Z 1369.556,A 0.000,B 0.000,C 90.000,E1 280.141} C_DIS
LIN {X 0.077,Y -457.889,Z 1369.553,A 0.000,B 0.000,C 90.000,E1 279.613} C_DIS
LIN {X 0.103,Y -457.420,Z 1369.551,A 0.000,B 0.000,C 90.000,E1 279.095} C_DIS
LIN {X 0.200,Y -456.438,Z 1369.548,A 0.000,B 0.000,C 90.000,E1 278.568} C_DIS
LIN {X -0.226,Y -454.965,Z 1369.545,A 0.000,B 0.000,C 90.000,E1 278.106} C_DIS
LIN {X -0.203,Y -452.973,Z 1369.542,A 0.000,B 0.000,C 90.000,E1 277.587} C_DIS
LIN {X -0.188,Y -450.438,Z 1369.539,A 0.000,B 0.000,C 90.000,E1 277.068} C_DIS
LIN {X -0.139,Y -447.315,Z 1369.536,A 0.000,B 0.000,C 90.000,E1 276.543} C_DIS
LIN {X -0.160,Y -443.449,Z 1369.533,A 0.000,B 0.000,C 90.000,E1 276.024} C_DIS
LIN {X 0.016,Y -441.203,Z 1369.532,A 0.000,B 0.000,C 90.000,E1 275.739} C_DIS
LIN {X 0.009,Y -435.843,Z 1369.529,A 0.000,B 0.000,C 90.000,E1 275.220} C_DIS
LIN {X -0.158,Y -429.767,Z 1369.526,A 0.000,B 0.000,C 90.000,E1 274.759} C_DIS
LIN {X 0.104,Y -423.371,Z 1369.524,A 0.000,B 0.000,C 90.000,E1 274.302} C_DIS
LIN {X -0.026,Y -416.842,Z 1369.522,A 0.000,B 0.000,C 90.000,E1 273.955} C_DIS
LIN {X 0.117,Y -410.309,Z 1369.520,A 0.000,B 0.000,C 90.000,E1 273.612} C_DIS
LIN {X 0.073,Y -403.644,Z 1369.519,A 0.000,B 0.000,C 90.000,E1 273.326} C_DIS
LIN {X -0.180,Y -393.479,Z 1369.516,A 0.000,B 0.000,C 90.000,E1 272.980} C_DIS
LIN {X -0.028,Y -383.338,Z 1369.515,A 0.000,B 0.000,C 90.000,E1 272.636} C_DIS
LIN {X -0.089,Y -375.908,Z 1369.514,A 0.000,B 0.000,C 90.000,E1 272.465} C_DIS
LIN {X 0.067,Y -368.001,Z 1369.513,A 0.000,B 0.000,C 90.000,E1 272.293} C_DIS
LIN {X 0.112,Y -351.817,Z 1369.512,A 0.000,B 0.000,C 90.000,E1 272.064} C_DIS
LIN {X -0.092,Y -340.400,Z 1369.511,A 0.000,B 0.000,C 90.000,E1 272.007} C_DIS
LIN {X 0.065,Y -331.354,Z 1369.511,A 0.000,B 0.000,C 90.000,E1 271.949} C_DIS
LIN {X 0.003,Y -181.270,Z 1369.511,A 0.000,B 0.000,C 90.000,E1 271.949} C_DIS
LIN {X 0.079,Y -181.574,Z 1369.502,A 0.000,B 0.000,C 90.000,E1 270.401} C_DIS
LIN {X 0.040,Y -180.911,Z 1369.476,A 0.000,B 0.000,C 90.000,E1 265.698} C_DIS
LIN {X -0.082,Y -180.827,Z 1369.471,A 0.000,B 0.000,C 90.000,E1 264.894} C_DIS
LIN {X -0.003,Y -178.932,Z 1369.443,A 0.000,B 0.000,C 90.000,E1 259.803} C_DIS
LIN {X 0.036,Y -175.980,Z 1369.415,A 0.000,B 0.000,C 90.000,E1 254.700} C_DIS
LIN {X -0.019,Y -175.472,Z 1369.410,A 0.000,B 0.000,C 90.000,E1 253.866} C_DIS
LIN {X 0.037,Y -172.219,Z 1369.387,A 0.000,B 0.000,C 90.000,E1 249.571} C_DIS
LIN {X 0.016,Y -171.696,Z 1369.382,A 0.000,B 0.000,C 90.000,E1 248.720} C_DIS
LIN {X 0.090,Y -167.290,Z 1369.353,A 0.000,B 0.000,C 90.000,E1 243.512} C_DIS
LIN {X 0.023,Y -166.667,Z 1369.348,A 0.000,B 0.000,C 90.000,E1 242.666} C_DIS
LIN {X -0.062,Y -162.649,Z 1369.324,A 0.000,B 0.000,C 90.000,E1 238.329} C_DIS
LIN {X 0.001,Y -161.338,Z 1369.314,A 0.000,B 0.000,C 90.000,E1 236.548} C_DIS
LIN {X 0.044,Y -157.333,Z 1369.290,A 0.000,B 0.000,C 90.000,E1 232.110} C_DIS
LIN {X -0.023,Y -155.316,Z 1369.275,A 0.000,B 0.000,C 90.000,E1 229.461} C_DIS
LIN {X 0.015,Y -151.671,Z 1369.250,A 0.000,B 0.000,C 90.000,E1 224.960} C_DIS
LIN {X -0.044,Y -150.537,Z 1369.240,A 0.000,B 0.000,C 90.000,E1 223.176} C_DIS
LIN {X -0.011,Y -147.261,Z 1369.215,A 0.000,B 0.000,C 90.000,E1 218.624} C_DIS
LIN {X 0.045,Y -145.288,Z 1369.194,A 0.000,B 0.000,C 90.000,E1 214.945} C_DIS
LIN {X -0.045,Y -142.388,Z 1369.164,A 0.000,B 0.000,C 90.000,E1 209.461} C_DIS
LIN {X 0.001,Y -141.366,Z 1369.148,A 0.000,B 0.000,C 90.000,E1 206.668} C_DIS
LIN {X -0.021,Y -139.344,Z 1369.112,A 0.000,B 0.000,C 90.000,E1 200.174} C_DIS
LIN {X -0.015,Y -139.015,Z 1369.102,A 0.000,B 0.000,C 90.000,E1 198.308} C_DIS
LIN {X -0.019,Y -138.342,Z 1369.055,A 0.000,B 0.000,C 90.000,E1 189.905} C_DIS
LIN {X 0.000,Y -139.395,Z 1369.008,A 0.000,B 0.000,C 90.000,E1 181.489} C_DIS
LIN {X 0.054,Y -141.297,Z 1368.972,A 0.000,B 0.000,C 90.000,E1 174.951} C_DIS
LIN {X 0.011,Y -142.659,Z 1368.957,A 0.000,B 0.000,C 90.000,E1 172.186} C_DIS
LIN {X -0.039,Y -145.002,Z 1368.931,A 0.000,B 0.000,C 90.000,E1 167.589} C_DIS
LIN {X -0.050,Y -147.629,Z 1368.911,A 0.000,B 0.000,C 90.000,E1 163.921} C_DIS
LIN {X 0.029,Y -150.257,Z 1368.890,A 0.000,B 0.000,C 90.000,E1 160.242} C_DIS
LIN {X 0.043,Y -153.655,Z 1368.870,A 0.000,B 0.000,C 90.000,E1 156.613} C_DIS
LIN {X -0.041,Y -157.071,Z 1368.850,A 0.000,B 0.000,C 90.000,E1 153.050} C_DIS
LIN {X 0.038,Y -161.203,Z 1368.830,A 0.000,B 0.000,C 90.000,E1 149.459} C_DIS
LIN {X -0.014,Y -163.295,Z 1368.821,A 0.000,B 0.000,C 90.000,E1 147.709} C_DIS
LIN {X -0.004,Y -167.741,Z 1368.801,A 0.000,B 0.000,C 90.000,E1 144.196} C_DIS
LIN {X -0.092,Y -171.559,Z 1368.787,A 0.000,B 0.000,C 90.000,E1 141.618} C_DIS
LIN {X -0.050,Y -176.503,Z 1368.767,A 0.000,B 0.000,C 90.000,E1 138.162} C_DIS
LIN {X 0.075,Y -180.801,Z 1368.753,A 0.000,B 0.000,C 90.000,E1 135.567} C_DIS
LIN {X 0.060,Y -186.209,Z 1368.735,A 0.000,B 0.000,C 90.000,E1 132.204} C_DIS
LIN {X -0.001,Y -190.846,Z 1368.721,A 0.000,B 0.000,C 90.000,E1 129.725} C_DIS
LIN {X 0.033,Y -196.607,Z 1368.702,A 0.000,B 0.000,C 90.000,E1 126.423} C_DIS
LIN {X 0.004,Y -199.222,Z 1368.695,A 0.000,B 0.000,C 90.000,E1 125.105} C_DIS
LIN {X -0.041,Y -308.952,Z 1368.695,A 0.000,B 0.000,C 90.000,E1 125.105} C_DIS
LIN {X -0.184,Y -310.915,Z 1368.695,A 0.000,B 0.000,C 90.000,E1 125.105} C_DIS
LIN {X -0.086,Y -316.408,Z 1368.693,A 0.000,B 0.000,C 90.000,E1 124.818} C_DIS
LIN {X 0.092,Y -319.535,Z 1368.692,A 0.000,B 0.000,C 90.000,E1 124.485} C_DIS
LIN {X -0.195,Y -323.144,Z 1368.689,A 0.000,B 0.000,C 90.000,E1 123.992} C_DIS
LIN {X 0.065,Y -324.620,Z 1368.687,A 0.000,B 0.000,C 90.000,E1 123.627} C_DIS
LIN {X -0.188,Y -337.441,Z 1368.668,A 0.000,B 0.000,C 90.000,E1 120.207} C_DIS
LIN {X 0.099,Y -349.353,Z 1368.652,A 0.000,B 0.000,C 90.000,E1 117.385} C_DIS
LIN {X -0.077,Y -362.723,Z 1368.637,A 0.000,B 0.000,C 90.000,E1 114.695} C_DIS
LIN {X -0.104,Y -375.921,Z 1368.624,A 0.000,B 0.000,C 90.000,E1 112.333} C_DIS
LIN {X 0.067,Y -390.450,Z 1368.611,A 0.000,B 0.000,C 90.000,E1 109.993} C_DIS
LIN {X -0.167,Y -406.413,Z 1368.599,A 0.000,B 0.000,C 90.000,E1 107.764} C_DIS
LIN {X -0.126,Y -423.921,Z 1368.586,A 0.000,B 0.000,C 90.000,E1 105.552} C_DIS
LIN {X -0.167,Y -443.070,Z 1368.574,A 0.000,B 0.000,C 90.000,E1 103.411} C_DIS
LIN {X 0.153,Y -463.159,Z 1368.563,A 0.000,B 0.000,C 90.000,E1 101.366} C_DIS
LIN {X -0.135,Y -481.165,Z 1368.554,A 0.000,B 0.000,C 90.000,E1 99.782} C_DIS
LIN {X -0.112,Y -483.371,Z 1368.553,A 0.000,B 0.000,C 90.000,E1 99.557} C_DIS
LIN {X -0.204,Y -485.192,Z 1368.552,A 0.000,B 0.000,C 90.000,E1 99.321} C_DIS
LIN {X 0.182,Y -486.563,Z 1368.550,A 0.000,B 0.000,C 90.000,E1 99.029} C_DIS
LIN {X -0.109,Y -488.306,Z 1368.547,A 0.000,B 0.000,C 90.000,E1 98.568} C_DIS
LIN {X 0.091,Y -488.953,Z 1368.545,A 0.000,B 0.000,C 90.000,E1 98.049} C_DIS
LIN {X -0.181,Y -488.615,Z 1368.542,A 0.000,B 0.000,C 90.000,E1 97.587} C_DIS
LIN {X 0.036,Y -487.241,Z 1368.539,A 0.000,B 0.000,C 90.000,E1 97.068} C_DIS
LIN {X -0.069,Y -486.096,Z 1368.538,A 0.000,B 0.000,C 90.000,E1 96.834} C_DIS
LIN {X -0.230,Y -484.563,Z 1368.536,A 0.000,B 0.000,C 90.000,E1 96.606} C_DIS
LIN {X -0.169,Y -474.052,Z 1368.528,A 0.000,B 0.000,C 90.000,E1 95.106} C_DIS
LIN {X -0.071,Y -462.634,Z 1368.518,A 0.000,B 0.000,C 90.000,E1 93.326} C_DIS
LIN {X -0.081,Y -442.889,Z 1368.501,A 0.000,B 0.000,C 90.000,E1 90.229} C_DIS
LIN {X -0.159,Y -427.986,Z 1368.486,A 0.000,B 0.000,C 90.000,E1 87.593} C_DIS
LIN {X 0.179,Y -419.143,Z 1368.478,A 0.000,B 0.000,C 90.000,E1 85.931} C_DIS
LIN {X 0.072,Y -408.666,Z 1368.467,A 0.000,B 0.000,C 90.000,E1 84.033} C_DIS
LIN {X 0.163,Y -399.563,Z 1368.458,A 0.000,B 0.000,C 90.000,E1 82.356} C_DIS
LIN {X 0.095,Y -390.250,Z 1368.448,A 0.000,B 0.000,C 90.000,E1 80.679} C_DIS
LIN {X -0.053,Y -379.165,Z 1368.437,A 0.000,B 0.000,C 90.000,E1 78.701} C_DIS
LIN {X 0.099,Y -369.486,Z 1368.427,A 0.000,B 0.000,C 90.000,E1 76.937} C_DIS
LIN {X 0.072,Y -359.658,Z 1368.418,A 0.000,B 0.000,C 90.000,E1 75.172} C_DIS
LIN {X 0.053,Y -349.722,Z 1368.408,A 0.000,B 0.000,C 90.000,E1 73.378} C_DIS
LIN {X -0.133,Y -337.996,Z 1368.396,A 0.000,B 0.000,C 90.000,E1 71.275} C_DIS
LIN {X -0.067,Y -324.710,Z 1368.382,A 0.000,B 0.000,C 90.000,E1 68.773} C_DIS
LIN {X 0.074,Y -307.440,Z 1368.362,A 0.000,B 0.000,C 90.000,E1 65.229} C_DIS
LIN {X 0.011,Y -296.256,Z 1368.348,A 0.000,B 0.000,C 90.000,E1 62.615} C_DIS
LIN {X -0.048,Y -286.283,Z 1368.333,A 0.000,B 0.000,C 90.000,E1 59.950} C_DIS
LIN {X -0.115,Y -278.523,Z 1368.320,A 0.000,B 0.000,C 90.000,E1 57.582} C_DIS
LIN {X -0.063,Y -268.414,Z 1368.301,A 0.000,B 0.000,C 90.000,E1 54.116} C_DIS
LIN {X -0.024,Y -260.707,Z 1368.285,A 0.000,B 0.000,C 90.000,E1 51.295} C_DIS
LIN {X -0.050,Y -253.373,Z 1368.269,A 0.000,B 0.000,C 90.000,E1 48.447} C_DIS
LIN {X -0.116,Y -244.669,Z 1368.249,A 0.000,B 0.000,C 90.000,E1 44.838} C_DIS
LIN {X -0.104,Y -236.827,Z 1368.229,A 0.000,B 0.000,C 90.000,E1 41.148} C_DIS
LIN {X 0.060,Y -229.840,Z 1368.208,A 0.000,B 0.000,C 90.000,E1 37.363} C_DIS
LIN {X 0.002,Y -223.775,Z 1368.187,A 0.000,B 0.000,C 90.000,E1 33.579} C_DIS
LIN {X -0.042,Y -218.600,Z 1368.165,A 0.000,B 0.000,C 90.000,E1 29.745} C_DIS
LIN {X -0.046,Y -213.753,Z 1368.139,A 0.000,B 0.000,C 90.000,E1 25.079} C_DIS
LIN {X -0.038,Y -209.781,Z 1368.109,A 0.000,B 0.000,C 90.000,E1 19.577} C_DIS
LIN {X 0.011,Y -207.558,Z 1368.087,A 0.000,B 0.000,C 90.000,E1 15.607} C_DIS
LIN {X -0.084,Y -205.493,Z 1368.065,A 0.000,B 0.000,C 90.000,E1 11.658} C_DIS
LIN {X -0.005,Y -203.650,Z 1368.042,A 0.000,B 0.000,C 90.000,E1 7.644} C_DIS
LIN {X 0.074,Y -202.364,Z 1368.025,A 0.000,B 0.000,C 90.000,E1 4.416} C_DIS
LIN {X 0.000,Y -200.857,Z 1368.000,A 0.000,B 0.000,C 90.000,E1 360.000} C_DIS
LIN {X 0.089,Y -199.904,Z 1367.970,A 0.000,B 0.000,C 90.000,E1 354.666} C_DIS
LIN {X 0.003,Y -200.335,Z 1367.935,A 0.000,B 0.000,C 90.000,E1 348.229} C_DIS
LIN {X 0.070,Y -202.866,Z 1367.899,A 0.000,B 0.000,C 90.000,E1 341.764} C_DIS
LIN {X 0.010,Y -206.231,Z 1367.872,A 0.000,B 0.000,C 90.000,E1 336.975} C_DIS
LIN {X 0.006,Y -210.243,Z 1367.850,A 0.000,B 0.000,C 90.000,E1 332.999} C_DIS
LIN {X -0.054,Y -215.431,Z 1367.828,A 0.000,B 0.000,C 90.000,E1 329.076} C_DIS
LIN {X -0.059,Y -221.892,Z 1367.807,A 0.000,B 0.000,C 90.000,E1 325.182} C_DIS
LIN {X -0.079,Y -227.840,Z 1367.789,A 0.000,B 0.000,C 90.000,E1 322.110} C_DIS
LIN {X -0.020,Y -234.735,Z 1367.772,A 0.000,B 0.000,C 90.000,E1 319.057} C_DIS
LIN {X -0.005,Y -243.392,Z 1367.754,A 0.000,B 0.000,C 90.000,E1 315.688} C_DIS
LIN {X 0.093,Y -253.123,Z 1367.735,A 0.000,B 0.000,C 90.000,E1 312.366} C_DIS
LIN {X 0.078,Y -261.788,Z 1367.721,A 0.000,B 0.000,C 90.000,E1 309.850} C_DIS
LIN {X 0.122,Y -271.415,Z 1367.708,A 0.000,B 0.000,C 90.000,E1 307.363} C_DIS
LIN {X 0.058,Y -282.067,Z 1367.694,A 0.000,B 0.000,C 90.000,E1 304.945} C_DIS
LIN {X 0.164,Y -292.430,Z 1367.683,A 0.000,B 0.000,C 90.000,E1 302.880} C_DIS
LIN {X -0.114,Y -302.086,Z 1367.674,A 0.000,B 0.000,C 90.000,E1 301.258} C_DIS
LIN {X -0.022,Y -310.924,Z 1367.666,A 0.000,B 0.000,C 90.000,E1 299.922} C_DIS
LIN {X 0.158,Y -320.501,Z 1367.659,A 0.000,B 0.000,C 90.000,E1 298.615} C_DIS
LIN {X 0.035,Y -344.355,Z 1367.644,A 0.000,B 0.000,C 90.000,E1 295.848} C_DIS
LIN {X 0.052,Y -357.616,Z 1367.635,A 0.000,B 0.000,C 90.000,E1 294.387} C_DIS
LIN {X -0.018,Y -370.737,Z 1367.627,A 0.000,B 0.000,C 90.000,E1 292.950} C_DIS
LIN {X 0.115,Y -383.514,Z 1367.619,A 0.000,B 0.000,C 90.000,E1 291.482} C_DIS
LIN {X -0.010,Y -395.952,Z 1367.611,A 0.000,B 0.000,C 90.000,E1 290.066} C_DIS
LIN {X -0.056,Y -413.170,Z 1367.601,A 0.000,B 0.000,C 90.000,E1 288.109} C_DIS
LIN {X -0.222,Y -422.937,Z 1367.594,A 0.000,B 0.000,C 90.000,E1 287.040} C_DIS
LIN {X -0.067,Y -429.800,Z 1367.590,A 0.000,B 0.000,C 90.000,E1 286.205} C_DIS
LIN {X 0.148,Y -436.103,Z 1367.585,A 0.000,B 0.000,C 90.000,E1 285.371} C_DIS
LIN {X 0.005,Y -441.715,Z 1367.581,A 0.000,B 0.000,C 90.000,E1 284.592} C_DIS
LIN {X -0.210,Y -446.514,Z 1367.577,A 0.000,B 0.000,C 90.000,E1 283.828} C_DIS
LIN {X -0.182,Y -449.279,Z 1367.574,A 0.000,B 0.000,C 90.000,E1 283.300} C_DIS
LIN {X -0.134,Y -451.699,Z 1367.571,A 0.000,B 0.000,C 90.000,E1 282.771} C_DIS
LIN {X -0.072,Y -453.769,Z 1367.568,A 0.000,B 0.000,C 90.000,E1 282.243} C_DIS
LIN {X 0.005,Y -455.474,Z 1367.565,A 0.000,B 0.000,C 90.000,E1 281.715} C_DIS
LIN {X 0.086,Y -456.816,Z 1367.562,A 0.000,B 0.000,C 90.000,E1 281.186} C_DIS
LIN {X 0.177,Y -457.675,Z 1367.559,A 0.000,B 0.000,C 90.000,E1 280.658} C_DIS
LIN {X 0.192,Y -458.182,Z 1367.557,A 0.000,B 0.000,C 90.000,E1 280.141} C_DIS
LIN {X -0.159,Y -458.230,Z 1367.554,A 0.000,B 0.000,C 90.000,E1 279.670} C_DIS
LIN {X -0.132,Y -457.773,Z 1367.551,A 0.000,B 0.000,C 90.000,E1 279.151} C_DIS
LIN {X -0.033,Y -456.844,Z 1367.548,A 0.000,B 0.000,C 90.000,E1 278.624} C_DIS
LIN {X -0.005,Y -455.410,Z 1367.545,A 0.000,B 0.000,C 90.000,E1 278.106} C_DIS
LIN {X 0.019,Y -453.452,Z 1367.542,A 0.000,B 0.000,C 90.000,E1 277.587} C_DIS
LIN {X 0.035,Y -450.964,Z 1367.539,A 0.000,B 0.000,C 90.000,E1 277.068} C_DIS
LIN {X 0.035,Y -447.890,Z 1367.536,A 0.000,B 0.000,C 90.000,E1 276.549} C_DIS
LIN {X 0.019,Y -444.128,Z 1367.534,A 0.000,B 0.000,C 90.000,E1 276.030} C_DIS
LIN {X -0.016,Y -439.473,Z 1367.531,A 0.000,B 0.000,C 90.000,E1 275.511} C_DIS
LIN {X 0.191,Y -436.741,Z 1367.529,A 0.000,B 0.000,C 90.000,E1 275.220} C_DIS
LIN {X -0.076,Y -433.641,Z 1367.528,A 0.000,B 0.000,C 90.000,E1 274.992} C_DIS
LIN {X -0.039,Y -427.377,Z 1367.525,A 0.000,B 0.000,C 90.000,E1 274.531} C_DIS
LIN {X -0.030,Y -420.900,Z 1367.523,A 0.000,B 0.000,C 90.000,E1 274.131} C_DIS
LIN {X -0.026,Y -414.388,Z 1367.521,A 0.000,B 0.000,C 90.000,E1 273.784} C_DIS
LIN {X 0.091,Y -404.831,Z 1367.519,A 0.000,B 0.000,C 90.000,E1 273.326} C_DIS
LIN {X -0.186,Y -394.723,Z 1367.516,A 0.000,B 0.000,C 90.000,E1 272.980} C_DIS
LIN {X -0.042,Y -384.714,Z 1367.515,A 0.000,B 0.000,C 90.000,E1 272.636} C_DIS
LIN {X -0.103,Y -377.518,Z 1367.514,A 0.000,B 0.000,C 90.000,E1 272.465} C_DIS
LIN {X 0.025,Y -369.624,Z 1367.513,A 0.000,B 0.000,C 90.000,E1 272.293} C_DIS
LIN {X 0.095,Y -353.607,Z 1367.512,A 0.000,B 0.000,C 90.000,E1 272.064} C_DIS
LIN {X -0.113,Y -343.664,Z 1367.511,A 0.000,B 0.000,C 90.000,E1 272.007} C_DIS
LIN {X -0.071,Y -329.797,Z 1367.511,A 0.000,B 0.000,C 90.000,E1 271.949} C_DIS
LIN {X -0.062,Y -181.274,Z 1367.511,A 0.000,B 0.000,C 90.000,E1 271.949} C_DIS
LIN {X -0.090,Y -181.580,Z 1367.501,A 0.000,B 0.000,C 90.000,E1 270.229} C_DIS
LIN {X 0.080,Y -180.889,Z 1367.473,A 0.000,B 0.000,C 90.000,E1 265.122} C_DIS
LIN {X -0.037,Y -179.013,Z 1367.445,A 0.000,B 0.000,C 90.000,E1 260.095} C_DIS
LIN {X 0.057,Y -178.633,Z 1367.440,A 0.000,B 0.000,C 90.000,E1 259.218} C_DIS
LIN {X -0.045,Y -175.684,Z 1367.412,A 0.000,B 0.000,C 90.000,E1 254.157} C_DIS
LIN {X -0.034,Y -172.401,Z 1367.388,A 0.000,B 0.000,C 90.000,E1 249.880} C_DIS
LIN {X -0.017,Y -171.210,Z 1367.379,A 0.000,B 0.000,C 90.000,E1 248.156} C_DIS
LIN {X 0.033,Y -167.495,Z 1367.355,A 0.000,B 0.000,C 90.000,E1 243.819} C_DIS
LIN {X 0.041,Y -166.892,Z 1367.350,A 0.000,B 0.000,C 90.000,E1 242.948} C_DIS
LIN {X 0.032,Y -162.197,Z 1367.321,A 0.000,B 0.000,C 90.000,E1 237.709} C_DIS
LIN {X -0.001,Y -160.770,Z 1367.311,A 0.000,B 0.000,C 90.000,E1 235.960} C_DIS
LIN {X -0.029,Y -157.565,Z 1367.291,A 0.000,B 0.000,C 90.000,E1 232.431} C_DIS
LIN {X 0.005,Y -155.596,Z 1367.276,A 0.000,B 0.000,C 90.000,E1 229.747} C_DIS
LIN {X 0.056,Y -151.877,Z 1367.251,A 0.000,B 0.000,C 90.000,E1 225.243} C_DIS
LIN {X 0.069,Y -150.103,Z 1367.236,A 0.000,B 0.000,C 90.000,E1 222.528} C_DIS
LIN {X -0.014,Y -146.899,Z 1367.211,A 0.000,B 0.000,C 90.000,E1 218.016} C_DIS
LIN {X 0.006,Y -145.487,Z 1367.196,A 0.000,B 0.000,C 90.000,E1 215.264} C_DIS
LIN {X 0.006,Y -142.895,Z 1367.170,A 0.000,B 0.000,C 90.000,E1 210.669} C_DIS
LIN {X -0.063,Y -141.515,Z 1367.150,A 0.000,B 0.000,C 90.000,E1 207.001} C_DIS
LIN {X -0.019,Y -139.393,Z 1367.114,A 0.000,B 0.000,C 90.000,E1 200.482} C_DIS
LIN {X 0.032,Y -139.103,Z 1367.103,A 0.000,B 0.000,C 90.000,E1 198.598} C_DIS
LIN {X 0.024,Y -138.354,Z 1367.057,A 0.000,B 0.000,C 90.000,E1 190.197} C_DIS
LIN {X 0.017,Y -139.513,Z 1367.005,A 0.000,B 0.000,C 90.000,E1 180.859} C_DIS
LIN {X -0.043,Y -141.161,Z 1366.974,A 0.000,B 0.000,C 90.000,E1 175.298} C_DIS
LIN {X 0.069,Y -142.540,Z 1366.958,A 0.000,B 0.000,C 90.000,E1 172.470} C_DIS
LIN {X -0.004,Y -144.812,Z 1366.933,A 0.000,B 0.000,C 90.000,E1 167.881} C_DIS
LIN {X -0.017,Y -147.431,Z 1366.912,A 0.000,B 0.000,C 90.000,E1 164.212} C_DIS
LIN {X 0.012,Y -150.010,Z 1366.892,A 0.000,B 0.000,C 90.000,E1 160.550} C_DIS
LIN {X 0.019,Y -153.343,Z 1366.872,A 0.000,B 0.000,C 90.000,E1 156.922} C_DIS
LIN {X 0.000,Y -155.878,Z 1366.857,A 0.000,B 0.000,C 90.000,E1 154.229} C_DIS
LIN {X -0.034,Y -159.733,Z 1366.837,A 0.000,B 0.000,C 90.000,E1 150.667} C_DIS
LIN {X 0.032,Y -161.972,Z 1366.827,A 0.000,B 0.000,C 90.000,E1 148.869} C_DIS
LIN {X -0.083,Y -166.164,Z 1366.807,A 0.000,B 0.000,C 90.000,E1 145.388} C_DIS
LIN {X -0.089,Y -171.177,Z 1366.788,A 0.000,B 0.000,C 90.000,E1 141.904} C_DIS
LIN {X 0.077,Y -176.059,Z 1366.769,A 0.000,B 0.000,C 90.000,E1 138.405} C_DIS
LIN {X -0.059,Y -180.315,Z 1366.755,A 0.000,B 0.000,C 90.000,E1 135.891} C_DIS
LIN {X -0.088,Y -185.726,Z 1366.736,A 0.000,B 0.000,C 90.000,E1 132.528} C_DIS
LIN {X -0.037,Y -190.334,Z 1366.722,A 0.000,B 0.000,C 90.000,E1 130.011} C_DIS
LIN {X 0.011,Y -197.660,Z 1366.699,A 0.000,B 0.000,C 90.000,E1 125.884} C_DIS
LIN {X 0.022,Y -199.212,Z 1366.695,A 0.000,B 0.000,C 90.000,E1 125.105} C_DIS
LIN {X -0.018,Y -309.156,Z 1366.695,A 0.000,B 0.000,C 90.000,E1 125.105} C_DIS
LIN {X -0.174,Y -311.045,Z 1366.695,A 0.000,B 0.000,C 90.000,E1 125.105} C_DIS
LIN {X -0.026,Y -314.380,Z 1366.694,A 0.000,B 0.000,C 90.000,E1 124.945} C_DIS
LIN {X 0.006,Y -317.732,Z 1366.693,A 0.000,B 0.000,C 90.000,E1 124.692} C_DIS
LIN {X 0.049,Y -321.389,Z 1366.690,A 0.000,B 0.000,C 90.000,E1 124.246} C_DIS
LIN {X 0.133,Y -323.244,Z 1366.688,A 0.000,B 0.000,C 90.000,E1 123.913} C_DIS
LIN {X -0.051,Y -324.686,Z 1366.687,A 0.000,B 0.000,C 90.000,E1 123.627} C_DIS
LIN {X 0.166,Y -337.493,Z 1366.667,A 0.000,B 0.000,C 90.000,E1 120.129} C_DIS
LIN {X -0.014,Y -349.418,Z 1366.652,A 0.000,B 0.000,C 90.000,E1 117.385} C_DIS
LIN {X 0.141,Y -362.793,Z 1366.637,A 0.000,B 0.000,C 90.000,E1 114.643} C_DIS
LIN {X 0.131,Y -376.000,Z 1366.624,A 0.000,B 0.000,C 90.000,E1 112.280} C_DIS
LIN {X -0.049,Y -390.538,Z 1366.611,A 0.000,B 0.000,C 90.000,E1 109.993} C_DIS
LIN {X 0.227,Y -406.512,Z 1366.599,A 0.000,B 0.000,C 90.000,E1 107.692} C_DIS
LIN {X -0.133,Y -424.031,Z 1366.586,A 0.000,B 0.000,C 90.000,E1 105.536} C_DIS
LIN {X 0.144,Y -443.188,Z 1366.574,A 0.000,B 0.000,C 90.000,E1 103.355} C_DIS
LIN {X 0.037,Y -463.280,Z 1366.563,A 0.000,B 0.000,C 90.000,E1 101.366} C_DIS
LIN {X 0.208,Y -481.308,Z 1366.554,A 0.000,B 0.000,C 90.000,E1 99.726} C_DIS
LIN {X -0.253,Y -483.451,Z 1366.553,A 0.000,B 0.000,C 90.000,E1 99.557} C_DIS
LIN {X -0.159,Y -485.079,Z 1366.552,A 0.000,B 0.000,C 90.000,E1 99.321} C_DIS
LIN {X 0.209,Y -486.454,Z 1366.550,A 0.000,B 0.000,C 90.000,E1 99.029} C_DIS
LIN {X 0.020,Y -487.471,Z 1366.549,A 0.000,B 0.000,C 90.000,E1 98.803} C_DIS
LIN {X -0.191,Y -488.626,Z 1366.546,A 0.000,B 0.000,C 90.000,E1 98.333} C_DIS
LIN {X 0.013,Y -488.767,Z 1366.543,A 0.000,B 0.000,C 90.000,E1 97.814} C_DIS
LIN {X 0.225,Y -487.917,Z 1366.541,A 0.000,B 0.000,C 90.000,E1 97.296} C_DIS
LIN {X -0.044,Y -485.932,Z 1366.538,A 0.000,B 0.000,C 90.000,E1 96.834} C_DIS
LIN {X -0.208,Y -484.387,Z 1366.537,A 0.000,B 0.000,C 90.000,E1 96.606} C_DIS
LIN {X -0.149,Y -473.850,Z 1366.528,A 0.000,B 0.000,C 90.000,E1 95.106} C_DIS
LIN {X 0.154,Y -464.052,Z 1366.520,A 0.000,B 0.000,C 90.000,E1 93.555} C_DIS
LIN {X 0.043,Y -452.320,Z 1366.510,A 0.000,B 0.000,C 90.000,E1 91.776} C_DIS
LIN {X 0.035,Y -438.116,Z 1366.497,A 0.000,B 0.000,C 90.000,E1 89.427} C_DIS
LIN {X -0.019,Y -426.320,Z 1366.485,A 0.000,B 0.000,C 90.000,E1 87.306} C_DIS
LIN {X -0.104,Y -417.463,Z 1366.476,A 0.000,B 0.000,C 90.000,E1 85.698} C_DIS
LIN {X 0.175,Y -406.999,Z 1366.465,A 0.000,B 0.000,C 90.000,E1 83.742} C_DIS
LIN {X -0.208,Y -397.882,Z 1366.456,A 0.000,B 0.000,C 90.000,E1 82.129} C_DIS
LIN {X 0.142,Y -388.536,Z 1366.447,A 0.000,B 0.000,C 90.000,E1 80.387} C_DIS
LIN {X -0.040,Y -377.448,Z 1366.436,A 0.000,B 0.000,C 90.000,E1 78.409} C_DIS
LIN {X 0.079,Y -367.718,Z 1366.426,A 0.000,B 0.000,C 90.000,E1 76.645} C_DIS
LIN {X 0.071,Y -356.227,Z 1366.414,A 0.000,B 0.000,C 90.000,E1 74.574} C_DIS
LIN {X -0.006,Y -346.258,Z 1366.404,A 0.000,B 0.000,C 90.000,E1 72.779} C_DIS
LIN {X 0.156,Y -334.531,Z 1366.392,A 0.000,B 0.000,C 90.000,E1 70.604} C_DIS
LIN {X 0.126,Y -321.336,Z 1366.378,A 0.000,B 0.000,C 90.000,E1 68.103} C_DIS
LIN {X -0.044,Y -305.859,Z 1366.361,A 0.000,B 0.000,C 90.000,E1 64.921} C_DIS
LIN {X -0.006,Y -294.868,Z 1366.346,A 0.000,B 0.000,C 90.000,E1 62.281} C_DIS
LIN {X 0.046,Y -285.039,Z 1366.331,A 0.000,B 0.000,C 90.000,E1 59.587} C_DIS
LIN {X 0.152,Y -273.338,Z 1366.310,A 0.000,B 0.000,C 90.000,E1 55.801} C_DIS
LIN {X -0.012,Y -265.492,Z 1366.295,A 0.000,B 0.000,C 90.000,E1 53.050} C_DIS
LIN {X 0.006,Y -256.115,Z 1366.275,A 0.000,B 0.000,C 90.000,E1 49.504} C_DIS
LIN {X 0.036,Y -247.289,Z 1366.255,A 0.000,B 0.000,C 90.000,E1 45.891} C_DIS
LIN {X -0.051,Y -239.183,Z 1366.235,A 0.000,B 0.000,C 90.000,E1 42.243} C_DIS
LIN {X -0.020,Y -231.951,Z 1366.214,A 0.000,B 0.000,C 90.000,E1 38.508} C_DIS
LIN {X -0.071,Y -225.616,Z 1366.193,A 0.000,B 0.000,C 90.000,E1 34.739} C_DIS
LIN {X 0.055,Y -220.175,Z 1366.172,A 0.000,B 0.000,C 90.000,E1 30.875} C_DIS
LIN {X 0.059,Y -215.745,Z 1366.150,A 0.000,B 0.000,C 90.000,E1 27.001} C_DIS
LIN {X -0.038,Y -211.748,Z 1366.124,A 0.000,B 0.000,C 90.000,E1 22.333} C_DIS
LIN {X 0.034,Y -208.810,Z 1366.098,A 0.000,B 0.000,C 90.000,E1 17.583} C_DIS
LIN {X -0.012,Y -207.069,Z 1366.080,A 0.000,B 0.000,C 90.000,E1 14.426} C_DIS
LIN {X 0.036,Y -205.048,Z 1366.058,A 0.000,B 0.000,C 90.000,E1 10.433} C_DIS
LIN {X 0.064,Y -203.257,Z 1366.036,A 0.000,B 0.000,C 90.000,E1 6.429} C_DIS
LIN {X 0.098,Y -201.701,Z 1366.014,A 0.000,B 0.000,C 90.000,E1 2.407} C_DIS
LIN {X -0.076,Y -200.303,Z 1365.984,A 0.000,B 0.000,C 90.000,E1 357.135} C_DIS
LIN {X -0.085,Y -200.072,Z 1365.948,A 0.000,B 0.000,C 90.000,E1 350.679} C_DIS
LIN {X 0.065,Y -202.169,Z 1365.908,A 0.000,B 0.000,C 90.000,E1 343.378} C_DIS
LIN {X -0.046,Y -205.729,Z 1365.877,A 0.000,B 0.000,C 90.000,E1 337.794} C_DIS
LIN {X -0.069,Y -209.536,Z 1365.854,A 0.000,B 0.000,C 90.000,E1 333.819} C_DIS
LIN {X -0.065,Y -214.495,Z 1365.833,A 0.000,B 0.000,C 90.000,E1 329.871} C_DIS
LIN {X -0.035,Y -220.691,Z 1365.811,A 0.000,B 0.000,C 90.000,E1 325.960} C_DIS
LIN {X -0.034,Y -228.021,Z 1365.789,A 0.000,B 0.000,C 90.000,E1 322.110} C_DIS
LIN {X 0.032,Y -234.893,Z 1365.773,A 0.000,B 0.000,C 90.000,E1 319.057} C_DIS
LIN {X -0.121,Y -243.541,Z 1365.754,A 0.000,B 0.000,C 90.000,E1 315.729} C_DIS
LIN {X -0.023,Y -252.098,Z 1365.738,A 0.000,B 0.000,C 90.000,E1 312.771} C_DIS
LIN {X -0.065,Y -260.608,Z 1365.724,A 0.000,B 0.000,C 90.000,E1 310.253} C_DIS
LIN {X 0.124,Y -270.095,Z 1365.710,A 0.000,B 0.000,C 90.000,E1 307.729} C_DIS
LIN {X 0.029,Y -280.586,Z 1365.696,A 0.000,B 0.000,C 90.000,E1 305.311} C_DIS
LIN {X 0.136,Y -288.969,Z 1365.687,A 0.000,B 0.000,C 90.000,E1 303.579} C_DIS
LIN {X -0.033,Y -298.208,Z 1365.677,A 0.000,B 0.000,C 90.000,E1 301.926} C_DIS
LIN {X -0.007,Y -304.308,Z 1365.672,A 0.000,B 0.000,C 90.000,E1 300.924} C_DIS
LIN {X -0.038,Y -313.343,Z 1365.665,A 0.000,B 0.000,C 90.000,E1 299.617} C_DIS
LIN {X -0.069,Y -325.842,Z 1365.656,A 0.000,B 0.000,C 90.000,E1 298.025} C_DIS
LIN {X -0.066,Y -346.970,Z 1365.642,A 0.000,B 0.000,C 90.000,E1 295.591} C_DIS
LIN {X -0.104,Y -360.275,Z 1365.634,A 0.000,B 0.000,C 90.000,E1 294.131} C_DIS
LIN {X 0.148,Y -370.639,Z 1365.628,A 0.000,B 0.000,C 90.000,E1 292.950} C_DIS
LIN {X -0.041,Y -383.347,Z 1365.620,A 0.000,B 0.000,C 90.000,E1 291.535} C_DIS
LIN {X -0.177,Y -395.787,Z 1365.612,A 0.000,B 0.000,C 90.000,E1 290.120} C_DIS
LIN {X 0.026,Y -412.970,Z 1365.601,A 0.000,B 0.000,C 90.000,E1 288.127} C_DIS
LIN {X -0.041,Y -422.767,Z 1365.595,A 0.000,B 0.000,C 90.000,E1 287.040} C_DIS
LIN {X -0.139,Y -431.852,Z 1365.589,A 0.000,B 0.000,C 90.000,E1 285.969} C_DIS
LIN {X 0.102,Y -437.946,Z 1365.584,A 0.000,B 0.000,C 90.000,E1 285.134} C_DIS
LIN {X 0.189,Y -441.639,Z 1365.581,A 0.000,B 0.000,C 90.000,E1 284.592} C_DIS
LIN {X -0.025,Y -446.510,Z 1365.577,A 0.000,B 0.000,C 90.000,E1 283.828} C_DIS
LIN {X 0.004,Y -449.303,Z 1365.574,A 0.000,B 0.000,C 90.000,E1 283.300} C_DIS
LIN {X -0.136,Y -452.864,Z 1365.570,A 0.000,B 0.000,C 90.000,E1 282.535} C_DIS
LIN {X 0.194,Y -455.568,Z 1365.565,A 0.000,B 0.000,C 90.000,E1 281.715} C_DIS
LIN {X -0.171,Y -456.962,Z 1365.562,A 0.000,B 0.000,C 90.000,E1 281.243} C_DIS
LIN {X -0.081,Y -457.896,Z 1365.559,A 0.000,B 0.000,C 90.000,E1 280.715} C_DIS
LIN {X -0.067,Y -458.443,Z 1365.557,A 0.000,B 0.000,C 90.000,E1 280.197} C_DIS
LIN {X 0.035,Y -458.514,Z 1365.554,A 0.000,B 0.000,C 90.000,E1 279.670} C_DIS
LIN {X 0.063,Y -458.104,Z 1365.551,A 0.000,B 0.000,C 90.000,E1 279.151} C_DIS
LIN {X 0.165,Y -457.237,Z 1365.548,A 0.000,B 0.000,C 90.000,E1 278.624} C_DIS
LIN {X 0.193,Y -455.826,Z 1365.545,A 0.000,B 0.000,C 90.000,E1 278.106} C_DIS
LIN {X -0.232,Y -453.941,Z 1365.542,A 0.000,B 0.000,C 90.000,E1 277.644} C_DIS
LIN {X -0.212,Y -451.466,Z 1365.539,A 0.000,B 0.000,C 90.000,E1 277.125} C_DIS
LIN {X -0.208,Y -448.451,Z 1365.536,A 0.000,B 0.000,C 90.000,E1 276.606} C_DIS
LIN {X -0.220,Y -444.784,Z 1365.534,A 0.000,B 0.000,C 90.000,E1 276.087} C_DIS
LIN {X 0.189,Y -440.280,Z 1365.531,A 0.000,B 0.000,C 90.000,E1 275.511} C_DIS
LIN {X 0.131,Y -434.581,Z 1365.528,A 0.000,B 0.000,C 90.000,E1 274.992} C_DIS
LIN {X 0.094,Y -428.406,Z 1365.525,A 0.000,B 0.000,C 90.000,E1 274.531} C_DIS
LIN {X 0.049,Y -421.933,Z 1365.523,A 0.000,B 0.000,C 90.000,E1 274.131} C_DIS
LIN {X 0.111,Y -412.300,Z 1365.520,A 0.000,B 0.000,C 90.000,E1 273.612} C_DIS
LIN {X 0.038,Y -405.740,Z 1365.519,A 0.000,B 0.000,C 90.000,E1 273.326} C_DIS
LIN {X 0.138,Y -395.703,Z 1365.516,A 0.000,B 0.000,C 90.000,E1 272.922} C_DIS
LIN {X -0.167,Y -385.396,Z 1365.515,A 0.000,B 0.000,C 90.000,E1 272.636} C_DIS
LIN {X 0.102,Y -378.050,Z 1365.513,A 0.000,B 0.000,C 90.000,E1 272.407} C_DIS
LIN {X -0.158,Y -369.783,Z 1365.513,A 0.000,B 0.000,C 90.000,E1 272.293} C_DIS
LIN {X -0.069,Y -353.418,Z 1365.511,A 0.000,B 0.000,C 90.000,E1 272.064} C_DIS
LIN {X 0.075,Y -343.366,Z 1365.511,A 0.000,B 0.000,C 90.000,E1 271.949} C_DIS
LIN {X 0.154,Y -330.440,Z 1365.511,A 0.000,B 0.000,C 90.000,E1 271.892} C_DIS
LIN {X 0.065,Y -181.276,Z 1365.511,A 0.000,B 0.000,C 90.000,E1 271.892} C_DIS
LIN {X 0.045,Y -181.579,Z 1365.501,A 0.000,B 0.000,C 90.000,E1 270.172} C_DIS
LIN {X 0.033,Y -180.887,Z 1365.473,A 0.000,B 0.000,C 90.000,E1 265.122} C_DIS
LIN {X -0.084,Y -179.009,Z 1365.445,A 0.000,B 0.000,C 90.000,E1 260.095} C_DIS
LIN {X 0.010,Y -178.622,Z 1365.440,A 0.000,B 0.000,C 90.000,E1 259.218} C_DIS
LIN {X 0.078,Y -175.674,Z 1365.412,A 0.000,B 0.000,C 90.000,E1 254.102} C_DIS
LIN {X -0.079,Y -172.391,Z 1365.388,A 0.000,B 0.000,C 90.000,E1 249.880} C_DIS
LIN {X -0.062,Y -171.195,Z 1365.379,A 0.000,B 0.000,C 90.000,E1 248.156} C_DIS
LIN {X -0.011,Y -167.484,Z 1365.354,A 0.000,B 0.000,C 90.000,E1 243.819} C_DIS
LIN {X -0.003,Y -166.881,Z 1365.350,A 0.000,B 0.000,C 90.000,E1 242.948} C_DIS
LIN {X -0.011,Y -162.186,Z 1365.321,A 0.000,B 0.000,C 90.000,E1 237.709} C_DIS
LIN {X 0.046,Y -160.755,Z 1365.311,A 0.000,B 0.000,C 90.000,E1 235.928} C_DIS
LIN {X 0.025,Y -157.552,Z 1365.291,A 0.000,B 0.000,C 90.000,E1 232.396} C_DIS
LIN {X -0.037,Y -155.581,Z 1365.276,A 0.000,B 0.000,C 90.000,E1 229.747} C_DIS
LIN {X 0.014,Y -151.866,Z 1365.251,A 0.000,B 0.000,C 90.000,E1 225.243} C_DIS
LIN {X 0.028,Y -150.090,Z 1365.236,A 0.000,B 0.000,C 90.000,E1 222.528} C_DIS
LIN {X -0.054,Y -146.891,Z 1365.211,A 0.000,B 0.000,C 90.000,E1 218.016} C_DIS
LIN {X 0.050,Y -145.477,Z 1365.196,A 0.000,B 0.000,C 90.000,E1 215.231} C_DIS
LIN {X -0.033,Y -142.888,Z 1365.170,A 0.000,B 0.000,C 90.000,E1 210.669} C_DIS
LIN {X 0.024,Y -141.507,Z 1365.150,A 0.000,B 0.000,C 90.000,E1 206.950} C_DIS
LIN {X -0.059,Y -139.391,Z 1365.114,A 0.000,B 0.000,C 90.000,E1 200.482} C_DIS
LIN {X -0.007,Y -139.098,Z 1365.103,A 0.000,B 0.000,C 90.000,E1 198.598} C_DIS
LIN {X -0.016,Y -138.354,Z 1365.057,A 0.000,B 0.000,C 90.000,E1 190.197} C_DIS
LIN {X -0.023,Y -139.515,Z 1365.005,A 0.000,B 0.000,C 90.000,E1 180.859} C_DIS
LIN {X 0.058,Y -141.168,Z 1364.974,A 0.000,B 0.000,C 90.000,E1 175.241} C_DIS
LIN {X 0.029,Y -142.547,Z 1364.958,A 0.000,B 0.000,C 90.000,E1 172.470} C_DIS
LIN {X -0.045,Y -144.822,Z 1364.933,A 0.000,B 0.000,C 90.000,E1 167.881} C_DIS
LIN {X -0.058,Y -147.443,Z 1364.912,A 0.000,B 0.000,C 90.000,E1 164.212} C_DIS
LIN {X -0.030,Y -150.024,Z 1364.892,A 0.000,B 0.000,C 90.000,E1 160.550} C_DIS
LIN {X -0.024,Y -153.360,Z 1364.872,A 0.000,B 0.000,C 90.000,E1 156.922} C_DIS
LIN {X 0.025,Y -155.893,Z 1364.857,A 0.000,B 0.000,C 90.000,E1 154.204} C_DIS
LIN {X -0.077,Y -159.751,Z 1364.837,A 0.000,B 0.000,C 90.000,E1 150.667} C_DIS
LIN {X -0.011,Y -161.991,Z 1364.827,A 0.000,B 0.000,C 90.000,E1 148.869} C_DIS
LIN {X 0.009,Y -166.184,Z 1364.807,A 0.000,B 0.000,C 90.000,E1 145.341} C_DIS
LIN {X 0.107,Y -171.199,Z 1364.788,A 0.000,B 0.000,C 90.000,E1 141.823} C_DIS
LIN {X 0.031,Y -176.081,Z 1364.769,A 0.000,B 0.000,C 90.000,E1 138.405} C_DIS
LIN {X -0.107,Y -180.342,Z 1364.755,A 0.000,B 0.000,C 90.000,E1 135.891} C_DIS
LIN {X 0.001,Y -185.752,Z 1364.736,A 0.000,B 0.000,C 90.000,E1 132.486} C_DIS
LIN {X -0.085,Y -190.363,Z 1364.722,A 0.000,B 0.000,C 90.000,E1 130.011} C_DIS
LIN {X -0.039,Y -197.689,Z 1364.699,A 0.000,B 0.000,C 90.000,E1 125.884} C_DIS
LIN {X 0.025,Y -199.209,Z 1364.695,A 0.000,B 0.000,C 90.000,E1 125.105} C_DIS
LIN {X 0.004,Y -309.141,Z 1364.695,A 0.000,B 0.000,C 90.000,E1 125.105} C_DIS
LIN {X 0.182,Y -311.691,Z 1364.695,A 0.000,B 0.000,C 90.000,E1 125.025} C_DIS
LIN {X 0.094,Y -314.849,Z 1364.694,A 0.000,B 0.000,C 90.000,E1 124.898} C_DIS
LIN {X 0.121,Y -318.345,Z 1364.692,A 0.000,B 0.000,C 90.000,E1 124.612} C_DIS
LIN {X -0.201,Y -321.966,Z 1364.690,A 0.000,B 0.000,C 90.000,E1 124.199} C_DIS
LIN {X 0.054,Y -323.690,Z 1364.688,A 0.000,B 0.000,C 90.000,E1 123.833} C_DIS
LIN {X -0.048,Y -326.132,Z 1364.684,A 0.000,B 0.000,C 90.000,E1 123.214} C_DIS
LIN {X -0.056,Y -336.603,Z 1364.669,A 0.000,B 0.000,C 90.000,E1 120.384} C_DIS
LIN {X 0.039,Y -348.414,Z 1364.653,A 0.000,B 0.000,C 90.000,E1 117.590} C_DIS
LIN {X -0.158,Y -361.676,Z 1364.638,A 0.000,B 0.000,C 90.000,E1 114.899} C_DIS
LIN {X -0.061,Y -374.771,Z 1364.625,A 0.000,B 0.000,C 90.000,E1 112.514} C_DIS
LIN {X 0.078,Y -389.190,Z 1364.612,A 0.000,B 0.000,C 90.000,E1 110.174} C_DIS
LIN {X -0.186,Y -405.034,Z 1364.600,A 0.000,B 0.000,C 90.000,E1 107.946} C_DIS
LIN {X -0.066,Y -422.413,Z 1364.587,A 0.000,B 0.000,C 90.000,E1 105.717} C_DIS
LIN {X 0.153,Y -441.448,Z 1364.575,A 0.000,B 0.000,C 90.000,E1 103.536} C_DIS
LIN {X 0.023,Y -461.490,Z 1364.564,A 0.000,B 0.000,C 90.000,E1 101.535} C_DIS
LIN {X 0.116,Y -481.976,Z 1364.554,A 0.000,B 0.000,C 90.000,E1 99.670} C_DIS
LIN {X 0.094,Y -483.954,Z 1364.552,A 0.000,B 0.000,C 90.000,E1 99.443} C_DIS
LIN {X 0.153,Y -485.461,Z 1364.551,A 0.000,B 0.000,C 90.000,E1 99.208} C_DIS
LIN {X 0.042,Y -486.704,Z 1364.550,A 0.000,B 0.000,C 90.000,E1 98.973} C_DIS
LIN {X -0.145,Y -487.612,Z 1364.548,A 0.000,B 0.000,C 90.000,E1 98.746} C_DIS
LIN {X 0.129,Y -488.585,Z 1364.546,A 0.000,B 0.000,C 90.000,E1 98.219} C_DIS
LIN {X -0.149,Y -488.558,Z 1364.543,A 0.000,B 0.000,C 90.000,E1 97.757} C_DIS
LIN {X 0.065,Y -487.530,Z 1364.540,A 0.000,B 0.000,C 90.000,E1 97.239} C_DIS
LIN {X -0.041,Y -486.593,Z 1364.539,A 0.000,B 0.000,C 90.000,E1 97.004} C_DIS
LIN {X -0.205,Y -485.319,Z 1364.537,A 0.000,B 0.000,C 90.000,E1 96.777} C_DIS
LIN {X 0.004,Y -471.489,Z 1364.526,A 0.000,B 0.000,C 90.000,E1 94.759} C_DIS
LIN {X -0.233,Y -461.610,Z 1364.518,A 0.000,B 0.000,C 90.000,E1 93.269} C_DIS
LIN {X -0.084,Y -440.425,Z 1364.499,A 0.000,B 0.000,C 90.000,E1 89.885} C_DIS
LIN {X 0.061,Y -427.112,Z 1364.486,A 0.000,B 0.000,C 90.000,E1 87.478} C_DIS
LIN {X -0.010,Y -418.286,Z 1364.477,A 0.000,B 0.000,C 90.000,E1 85.869} C_DIS
LIN {X -0.057,Y -406.339,Z 1364.465,A 0.000,B 0.000,C 90.000,E1 83.685} C_DIS
LIN {X 0.001,Y -397.215,Z 1364.456,A 0.000,B 0.000,C 90.000,E1 82.008} C_DIS
LIN {X -0.105,Y -387.880,Z 1364.446,A 0.000,B 0.000,C 90.000,E1 80.330} C_DIS
LIN {X 0.149,Y -376.790,Z 1364.435,A 0.000,B 0.000,C 90.000,E1 78.285} C_DIS
LIN {X -0.185,Y -367.068,Z 1364.425,A 0.000,B 0.000,C 90.000,E1 76.589} C_DIS
LIN {X -0.201,Y -355.568,Z 1364.414,A 0.000,B 0.000,C 90.000,E1 74.519} C_DIS
LIN {X 0.044,Y -345.582,Z 1364.404,A 0.000,B 0.000,C 90.000,E1 72.670} C_DIS
LIN {X -0.142,Y -332.207,Z 1364.390,A 0.000,B 0.000,C 90.000,E1 70.242} C_DIS
LIN {X 0.138,Y -317.496,Z 1364.374,A 0.000,B 0.000,C 90.000,E1 67.358} C_DIS
LIN {X 0.088,Y -303.838,Z 1364.358,A 0.000,B 0.000,C 90.000,E1 64.460} C_DIS
LIN {X 0.074,Y -294.356,Z 1364.345,A 0.000,B 0.000,C 90.000,E1 62.153} C_DIS
LIN {X 0.135,Y -285.726,Z 1364.332,A 0.000,B 0.000,C 90.000,E1 59.793} C_DIS
LIN {X -0.130,Y -277.050,Z 1364.317,A 0.000,B 0.000,C 90.000,E1 57.120} C_DIS
LIN {X 0.025,Y -267.110,Z 1364.298,A 0.000,B 0.000,C 90.000,E1 53.623} C_DIS
LIN {X -0.072,Y -257.662,Z 1364.278,A 0.000,B 0.000,C 90.000,E1 50.114} C_DIS
LIN {X 0.011,Y -248.758,Z 1364.258,A 0.000,B 0.000,C 90.000,E1 46.500} C_DIS
LIN {X -0.032,Y -240.530,Z 1364.238,A 0.000,B 0.000,C 90.000,E1 42.852} C_DIS
LIN {X 0.042,Y -233.214,Z 1364.217,A 0.000,B 0.000,C 90.000,E1 39.116} C_DIS
LIN {X -0.017,Y -226.715,Z 1364.196,A 0.000,B 0.000,C 90.000,E1 35.358} C_DIS
LIN {X -0.047,Y -221.137,Z 1364.175,A 0.000,B 0.000,C 90.000,E1 31.544} C_DIS
LIN {X 0.093,Y -216.544,Z 1364.154,A 0.000,B 0.000,C 90.000,E1 27.641} C_DIS
LIN {X 0.109,Y -212.378,Z 1364.128,A 0.000,B 0.000,C 90.000,E1 22.950} C_DIS
LIN {X 0.072,Y -209.336,Z 1364.101,A 0.000,B 0.000,C 90.000,E1 18.236} C_DIS
LIN {X -0.017,Y -207.110,Z 1364.079,A 0.000,B 0.000,C 90.000,E1 14.300} C_DIS
LIN {X 0.024,Y -205.089,Z 1364.057,A 0.000,B 0.000,C 90.000,E1 10.310} C_DIS
LIN {X 0.020,Y -203.288,Z 1364.035,A 0.000,B 0.000,C 90.000,E1 6.315} C_DIS
LIN {X 0.057,Y -201.724,Z 1364.013,A 0.000,B 0.000,C 90.000,E1 2.293} C_DIS
LIN {X -0.084,Y -200.248,Z 1363.979,A 0.000,B 0.000,C 90.000,E1 356.331} C_DIS
LIN {X -0.037,Y -200.268,Z 1363.944,A 0.000,B 0.000,C 90.000,E1 349.859} C_DIS
LIN {X -0.010,Y -202.714,Z 1363.903,A 0.000,B 0.000,C 90.000,E1 342.598} C_DIS
LIN {X -0.028,Y -205.892,Z 1363.877,A 0.000,B 0.000,C 90.000,E1 337.794} C_DIS
LIN {X -0.046,Y -209.705,Z 1363.854,A 0.000,B 0.000,C 90.000,E1 333.819} C_DIS
LIN {X -0.036,Y -214.676,Z 1363.833,A 0.000,B 0.000,C 90.000,E1 329.871} C_DIS
LIN {X 0.001,Y -220.874,Z 1363.811,A 0.000,B 0.000,C 90.000,E1 325.960} C_DIS
LIN {X 0.009,Y -228.196,Z 1363.790,A 0.000,B 0.000,C 90.000,E1 322.110} C_DIS
LIN {X -0.074,Y -235.051,Z 1363.773,A 0.000,B 0.000,C 90.000,E1 319.094} C_DIS
LIN {X -0.066,Y -243.690,Z 1363.754,A 0.000,B 0.000,C 90.000,E1 315.729} C_DIS
LIN {X 0.038,Y -252.225,Z 1363.738,A 0.000,B 0.000,C 90.000,E1 312.771} C_DIS
LIN {X 0.001,Y -260.730,Z 1363.724,A 0.000,B 0.000,C 90.000,E1 310.253} C_DIS
LIN {X -0.184,Y -270.221,Z 1363.710,A 0.000,B 0.000,C 90.000,E1 307.810} C_DIS
LIN {X 0.105,Y -280.701,Z 1363.696,A 0.000,B 0.000,C 90.000,E1 305.311} C_DIS
LIN {X -0.024,Y -289.075,Z 1363.687,A 0.000,B 0.000,C 90.000,E1 303.627} C_DIS
LIN {X 0.052,Y -298.320,Z 1363.677,A 0.000,B 0.000,C 90.000,E1 301.926} C_DIS
LIN {X 0.100,Y -306.602,Z 1363.670,A 0.000,B 0.000,C 90.000,E1 300.590} C_DIS
LIN {X 0.102,Y -315.847,Z 1363.663,A 0.000,B 0.000,C 90.000,E1 299.283} C_DIS
LIN {X 0.001,Y -333.890,Z 1363.650,A 0.000,B 0.000,C 90.000,E1 297.078} C_DIS
LIN {X -0.056,Y -349.886,Z 1363.640,A 0.000,B 0.000,C 90.000,E1 295.283} C_DIS
LIN {X -0.083,Y -363.171,Z 1363.632,A 0.000,B 0.000,C 90.000,E1 293.823} C_DIS
LIN {X -0.016,Y -370.980,Z 1363.627,A 0.000,B 0.000,C 90.000,E1 292.950} C_DIS
LIN {X 0.111,Y -383.717,Z 1363.619,A 0.000,B 0.000,C 90.000,E1 291.482} C_DIS
LIN {X -0.005,Y -396.128,Z 1363.611,A 0.000,B 0.000,C 90.000,E1 290.066} C_DIS
LIN {X 0.127,Y -410.801,Z 1363.602,A 0.000,B 0.000,C 90.000,E1 288.362} C_DIS
LIN {X 0.014,Y -420.685,Z 1363.596,A 0.000,B 0.000,C 90.000,E1 287.275} C_DIS
LIN {X 0.142,Y -427.697,Z 1363.591,A 0.000,B 0.000,C 90.000,E1 286.441} C_DIS
LIN {X -0.071,Y -434.235,Z 1363.587,A 0.000,B 0.000,C 90.000,E1 285.662} C_DIS
LIN {X 0.184,Y -440.121,Z 1363.583,A 0.000,B 0.000,C 90.000,E1 284.828} C_DIS
LIN {X -0.038,Y -445.252,Z 1363.578,A 0.000,B 0.000,C 90.000,E1 284.064} C_DIS
LIN {X -0.017,Y -448.255,Z 1363.575,A 0.000,B 0.000,C 90.000,E1 283.536} C_DIS
LIN {X -0.172,Y -452.026,Z 1363.571,A 0.000,B 0.000,C 90.000,E1 282.771} C_DIS
LIN {X -0.107,Y -454.109,Z 1363.568,A 0.000,B 0.000,C 90.000,E1 282.243} C_DIS
LIN {X -0.029,Y -455.817,Z 1363.565,A 0.000,B 0.000,C 90.000,E1 281.715} C_DIS
LIN {X 0.055,Y -457.187,Z 1363.562,A 0.000,B 0.000,C 90.000,E1 281.186} C_DIS
LIN {X 0.147,Y -458.192,Z 1363.559,A 0.000,B 0.000,C 90.000,E1 280.658} C_DIS
LIN {X 0.164,Y -458.709,Z 1363.556,A 0.000,B 0.000,C 90.000,E1 280.141} C_DIS
LIN {X -0.184,Y -458.813,Z 1363.554,A 0.000,B 0.000,C 90.000,E1 279.670} C_DIS
LIN {X -0.154,Y -458.394,Z 1363.551,A 0.000,B 0.000,C 90.000,E1 279.151} C_DIS
LIN {X -0.051,Y -457.508,Z 1363.548,A 0.000,B 0.000,C 90.000,E1 278.624} C_DIS
LIN {X -0.020,Y -456.135,Z 1363.545,A 0.000,B 0.000,C 90.000,E1 278.106} C_DIS
LIN {X 0.007,Y -454.221,Z 1363.542,A 0.000,B 0.000,C 90.000,E1 277.587} C_DIS
LIN {X 0.028,Y -451.727,Z 1363.539,A 0.000,B 0.000,C 90.000,E1 277.068} C_DIS
LIN {X 0.033,Y -448.663,Z 1363.536,A 0.000,B 0.000,C 90.000,E1 276.549} C_DIS
LIN {X 0.022,Y -445.021,Z 1363.534,A 0.000,B 0.000,C 90.000,E1 276.030} C_DIS
LIN {X -0.009,Y -440.552,Z 1363.531,A 0.000,B 0.000,C 90.000,E1 275.511} C_DIS
LIN {X -0.063,Y -434.887,Z 1363.528,A 0.000,B 0.000,C 90.000,E1 274.992} C_DIS
LIN {X -0.116,Y -428.733,Z 1363.525,A 0.000,B 0.000,C 90.000,E1 274.531} C_DIS
LIN {X -0.102,Y -422.419,Z 1363.523,A 0.000,B 0.000,C 90.000,E1 274.131} C_DIS
LIN {X -0.169,Y -415.922,Z 1363.521,A 0.000,B 0.000,C 90.000,E1 273.784} C_DIS
LIN {X -0.195,Y -406.087,Z 1363.518,A 0.000,B 0.000,C 90.000,E1 273.326} C_DIS
LIN {X -0.119,Y -395.928,Z 1363.516,A 0.000,B 0.000,C 90.000,E1 272.922} C_DIS
LIN {X -0.007,Y -385.743,Z 1363.514,A 0.000,B 0.000,C 90.000,E1 272.579} C_DIS
LIN {X -0.098,Y -378.430,Z 1363.513,A 0.000,B 0.000,C 90.000,E1 272.407} C_DIS
LIN {X 0.029,Y -370.167,Z 1363.512,A 0.000,B 0.000,C 90.000,E1 272.236} C_DIS
LIN {X -0.148,Y -349.311,Z 1363.511,A 0.000,B 0.000,C 90.000,E1 272.007} C_DIS
LIN {X 0.086,Y -335.143,Z 1363.511,A 0.000,B 0.000,C 90.000,E1 271.892} C_DIS
LIN {X 0.013,Y -181.279,Z 1363.510,A 0.000,B 0.000,C 90.000,E1 271.892} C_DIS
LIN {X 0.088,Y -181.578,Z 1363.502,A 0.000,B 0.000,C 90.000,E1 270.344} C_DIS
LIN {X -0.075,Y -180.809,Z 1363.471,A 0.000,B 0.000,C 90.000,E1 264.837} C_DIS
LIN {X 0.002,Y -178.911,Z 1363.443,A 0.000,B 0.000,C 90.000,E1 259.746} C_DIS
LIN {X 0.082,Y -175.955,Z 1363.415,A 0.000,B 0.000,C 90.000,E1 254.629} C_DIS
LIN {X 0.028,Y -175.424,Z 1363.410,A 0.000,B 0.000,C 90.000,E1 253.795} C_DIS
LIN {X 0.030,Y -172.185,Z 1363.386,A 0.000,B 0.000,C 90.000,E1 249.518} C_DIS
LIN {X 0.070,Y -171.656,Z 1363.381,A 0.000,B 0.000,C 90.000,E1 248.646} C_DIS
LIN {X 0.064,Y -167.881,Z 1363.358,A 0.000,B 0.000,C 90.000,E1 244.332} C_DIS
LIN {X 0.007,Y -166.617,Z 1363.348,A 0.000,B 0.000,C 90.000,E1 242.615} C_DIS
LIN {X 0.000,Y -162.605,Z 1363.324,A 0.000,B 0.000,C 90.000,E1 238.250} C_DIS
LIN {X -0.025,Y -161.289,Z 1363.314,A 0.000,B 0.000,C 90.000,E1 236.501} C_DIS
LIN {X 0.009,Y -157.288,Z 1363.289,A 0.000,B 0.000,C 90.000,E1 232.065} C_DIS
LIN {X 0.032,Y -156.006,Z 1363.279,A 0.000,B 0.000,C 90.000,E1 230.275} C_DIS
LIN {X -0.008,Y -152.264,Z 1363.255,A 0.000,B 0.000,C 90.000,E1 225.810} C_DIS
LIN {X 0.014,Y -150.501,Z 1363.240,A 0.000,B 0.000,C 90.000,E1 223.095} C_DIS
LIN {X 0.044,Y -147.226,Z 1363.214,A 0.000,B 0.000,C 90.000,E1 218.543} C_DIS
LIN {X 0.013,Y -145.248,Z 1363.194,A 0.000,B 0.000,C 90.000,E1 214.898} C_DIS
LIN {X -0.070,Y -142.365,Z 1363.163,A 0.000,B 0.000,C 90.000,E1 209.411} C_DIS
LIN {X 0.051,Y -141.751,Z 1363.153,A 0.000,B 0.000,C 90.000,E1 207.513} C_DIS
LIN {X -0.024,Y -139.494,Z 1363.117,A 0.000,B 0.000,C 90.000,E1 201.046} C_DIS
LIN {X 0.013,Y -138.998,Z 1363.101,A 0.000,B 0.000,C 90.000,E1 198.236} C_DIS
LIN {X -0.030,Y -138.337,Z 1363.055,A 0.000,B 0.000,C 90.000,E1 189.849} C_DIS
LIN {X -0.008,Y -139.411,Z 1363.008,A 0.000,B 0.000,C 90.000,E1 181.432} C_DIS
LIN {X 0.045,Y -141.324,Z 1362.972,A 0.000,B 0.000,C 90.000,E1 174.894} C_DIS
LIN {X 0.003,Y -142.682,Z 1362.956,A 0.000,B 0.000,C 90.000,E1 172.129} C_DIS
LIN {X -0.018,Y -145.039,Z 1362.931,A 0.000,B 0.000,C 90.000,E1 167.521} C_DIS
LIN {X -0.020,Y -147.666,Z 1362.910,A 0.000,B 0.000,C 90.000,E1 163.850} C_DIS
LIN {X 0.015,Y -150.307,Z 1362.890,A 0.000,B 0.000,C 90.000,E1 160.188} C_DIS
LIN {X 0.026,Y -153.718,Z 1362.870,A 0.000,B 0.000,C 90.000,E1 156.561} C_DIS
LIN {X -0.060,Y -157.131,Z 1362.850,A 0.000,B 0.000,C 90.000,E1 152.999} C_DIS
LIN {X 0.015,Y -161.277,Z 1362.830,A 0.000,B 0.000,C 90.000,E1 149.410} C_DIS
LIN {X 0.033,Y -164.395,Z 1362.815,A 0.000,B 0.000,C 90.000,E1 146.755} C_DIS
LIN {X 0.030,Y -169.073,Z 1362.796,A 0.000,B 0.000,C 90.000,E1 143.256} C_DIS
LIN {X -0.019,Y -171.631,Z 1362.786,A 0.000,B 0.000,C 90.000,E1 141.537} C_DIS
LIN {X 0.028,Y -176.591,Z 1362.767,A 0.000,B 0.000,C 90.000,E1 138.081} C_DIS
LIN {X -0.099,Y -180.889,Z 1362.753,A 0.000,B 0.000,C 90.000,E1 135.567} C_DIS
LIN {X 0.022,Y -186.305,Z 1362.734,A 0.000,B 0.000,C 90.000,E1 132.162} C_DIS
LIN {X 0.088,Y -190.938,Z 1362.720,A 0.000,B 0.000,C 90.000,E1 129.644} C_DIS
LIN {X 0.009,Y -196.708,Z 1362.702,A 0.000,B 0.000,C 90.000,E1 126.377} C_DIS
LIN {X 0.039,Y -199.201,Z 1362.695,A 0.000,B 0.000,C 90.000,E1 125.105} C_DIS
LIN {X 0.002,Y -309.531,Z 1362.695,A 0.000,B 0.000,C 90.000,E1 125.105} C_DIS
LIN {X 0.131,Y -314.760,Z 1362.694,A 0.000,B 0.000,C 90.000,E1 124.898} C_DIS
LIN {X 0.063,Y -317.111,Z 1362.693,A 0.000,B 0.000,C 90.000,E1 124.739} C_DIS
LIN {X -0.053,Y -320.955,Z 1362.691,A 0.000,B 0.000,C 90.000,E1 124.326} C_DIS
LIN {X 0.103,Y -322.828,Z 1362.689,A 0.000,B 0.000,C 90.000,E1 123.992} C_DIS
LIN {X -0.007,Y -324.291,Z 1362.687,A 0.000,B 0.000,C 90.000,E1 123.706} C_DIS
LIN {X 0.047,Y -338.363,Z 1362.666,A 0.000,B 0.000,C 90.000,E1 119.922} C_DIS
LIN {X 0.198,Y -350.396,Z 1362.651,A 0.000,B 0.000,C 90.000,E1 117.129} C_DIS
LIN {X -0.097,Y -363.898,Z 1362.636,A 0.000,B 0.000,C 90.000,E1 114.463} C_DIS
LIN {X 0.058,Y -377.221,Z 1362.623,A 0.000,B 0.000,C 90.000,E1 112.078} C_DIS
LIN {X 0.129,Y -391.887,Z 1362.610,A 0.000,B 0.000,C 90.000,E1 109.758} C_DIS
LIN {X 0.063,Y -407.996,Z 1362.597,A 0.000,B 0.000,C 90.000,E1 107.511} C_DIS
LIN {X 0.028,Y -425.663,Z 1362.585,A 0.000,B 0.000,C 90.000,E1 105.315} C_DIS
LIN {X 0.059,Y -444.954,Z 1362.573,A 0.000,B 0.000,C 90.000,E1 103.175} C_DIS
LIN {X 0.068,Y -465.100,Z 1362.562,A 0.000,B 0.000,C 90.000,E1 101.186} C_DIS
LIN {X 0.153,Y -480.561,Z 1362.554,A 0.000,B 0.000,C 90.000,E1 99.792} C_DIS
LIN {X -0.200,Y -482.803,Z 1362.553,A 0.000,B 0.000,C 90.000,E1 99.613} C_DIS
LIN {X -0.082,Y -484.501,Z 1362.552,A 0.000,B 0.000,C 90.000,E1 99.378} C_DIS
LIN {X 0.207,Y -485.955,Z 1362.551,A 0.000,B 0.000,C 90.000,E1 99.095} C_DIS
LIN {X 0.093,Y -487.036,Z 1362.549,A 0.000,B 0.000,C 90.000,E1 98.859} C_DIS
LIN {X -0.193,Y -488.298,Z 1362.547,A 0.000,B 0.000,C 90.000,E1 98.398} C_DIS
LIN {X 0.080,Y -488.533,Z 1362.544,A 0.000,B 0.000,C 90.000,E1 97.871} C_DIS
LIN {X -0.193,Y -487.783,Z 1362.541,A 0.000,B 0.000,C 90.000,E1 97.409} C_DIS
LIN {X 0.019,Y -485.922,Z 1362.538,A 0.000,B 0.000,C 90.000,E1 96.891} C_DIS
LIN {X -0.147,Y -484.463,Z 1362.537,A 0.000,B 0.000,C 90.000,E1 96.663} C_DIS
LIN {X 0.198,Y -472.202,Z 1362.527,A 0.000,B 0.000,C 90.000,E1 94.878} C_DIS
LIN {X 0.007,Y -462.313,Z 1362.519,A 0.000,B 0.000,C 90.000,E1 93.383} C_DIS
LIN {X -0.212,Y -444.173,Z 1362.503,A 0.000,B 0.000,C 90.000,E1 90.573} C_DIS
LIN {X 0.180,Y -429.190,Z 1362.488,A 0.000,B 0.000,C 90.000,E1 87.879} C_DIS
LIN {X -0.190,Y -418.925,Z 1362.478,A 0.000,B 0.000,C 90.000,E1 86.045} C_DIS
LIN {X -0.183,Y -406.994,Z 1362.466,A 0.000,B 0.000,C 90.000,E1 83.856} C_DIS
LIN {X -0.162,Y -397.907,Z 1362.456,A 0.000,B 0.000,C 90.000,E1 82.186} C_DIS
LIN {X 0.190,Y -388.599,Z 1362.447,A 0.000,B 0.000,C 90.000,E1 80.443} C_DIS
LIN {X 0.011,Y -377.513,Z 1362.436,A 0.000,B 0.000,C 90.000,E1 78.465} C_DIS
LIN {X 0.132,Y -367.834,Z 1362.426,A 0.000,B 0.000,C 90.000,E1 76.700} C_DIS
LIN {X 0.127,Y -356.323,Z 1362.415,A 0.000,B 0.000,C 90.000,E1 74.629} C_DIS
LIN {X 0.053,Y -346.372,Z 1362.405,A 0.000,B 0.000,C 90.000,E1 72.834} C_DIS
LIN {X 0.109,Y -334.657,Z 1362.393,A 0.000,B 0.000,C 90.000,E1 70.678} C_DIS
LIN {X 0.196,Y -321.460,Z 1362.379,A 0.000,B 0.000,C 90.000,E1 68.156} C_DIS
LIN {X 0.034,Y -305.982,Z 1362.361,A 0.000,B 0.000,C 90.000,E1 64.973} C_DIS
LIN {X 0.069,Y -296.260,Z 1362.348,A 0.000,B 0.000,C 90.000,E1 62.666} C_DIS
LIN {X 0.014,Y -286.279,Z 1362.333,A 0.000,B 0.000,C 90.000,E1 59.999} C_DIS
LIN {X -0.159,Y -279.645,Z 1362.322,A 0.000,B 0.000,C 90.000,E1 57.995} C_DIS
LIN {X 0.148,Y -269.546,Z 1362.303,A 0.000,B 0.000,C 90.000,E1 54.482} C_DIS
LIN {X 0.044,Y -261.886,Z 1362.287,A 0.000,B 0.000,C 90.000,E1 51.698} C_DIS
LIN {X 0.037,Y -254.560,Z 1362.271,A 0.000,B 0.000,C 90.000,E1 48.852} C_DIS
LIN {X 0.000,Y -245.863,Z 1362.251,A 0.000,B 0.000,C 90.000,E1 45.243} C_DIS
LIN {X 0.048,Y -237.992,Z 1362.231,A 0.000,B 0.000,C 90.000,E1 41.553} C_DIS
LIN {X 0.072,Y -230.948,Z 1362.210,A 0.000,B 0.000,C 90.000,E1 37.810} C_DIS
LIN {X -0.007,Y -224.786,Z 1362.189,A 0.000,B 0.000,C 90.000,E1 34.040} C_DIS
LIN {X -0.025,Y -219.551,Z 1362.168,A 0.000,B 0.000,C 90.000,E1 30.207} C_DIS
LIN {X 0.010,Y -214.613,Z 1362.142,A 0.000,B 0.000,C 90.000,E1 25.540} C_DIS
LIN {X -0.054,Y -210.570,Z 1362.111,A 0.000,B 0.000,C 90.000,E1 20.066} C_DIS
LIN {X 0.083,Y -208.223,Z 1362.089,A 0.000,B 0.000,C 90.000,E1 16.079} C_DIS
LIN {X 0.050,Y -206.090,Z 1362.067,A 0.000,B 0.000,C 90.000,E1 12.119} C_DIS
LIN {X 0.100,Y -204.522,Z 1362.050,A 0.000,B 0.000,C 90.000,E1 8.916} C_DIS
LIN {X 0.029,Y -202.792,Z 1362.027,A 0.000,B 0.000,C 90.000,E1 4.935} C_DIS
LIN {X 0.038,Y -201.318,Z 1362.005,A 0.000,B 0.000,C 90.000,E1 0.917} C_DIS
LIN {X -0.092,Y -200.208,Z 1361.975,A 0.000,B 0.000,C 90.000,E1 355.527} C_DIS
LIN {X -0.023,Y -200.513,Z 1361.939,A 0.000,B 0.000,C 90.000,E1 349.050} C_DIS
LIN {X 0.000,Y -202.850,Z 1361.903,A 0.000,B 0.000,C 90.000,E1 342.598} C_DIS
LIN {X -0.012,Y -206.040,Z 1361.877,A 0.000,B 0.000,C 90.000,E1 337.794} C_DIS
LIN {X 0.080,Y -210.748,Z 1361.850,A 0.000,B 0.000,C 90.000,E1 332.999} C_DIS
LIN {X 0.037,Y -216.000,Z 1361.828,A 0.000,B 0.000,C 90.000,E1 329.076} C_DIS
LIN {X 0.054,Y -222.416,Z 1361.807,A 0.000,B 0.000,C 90.000,E1 325.182} C_DIS
LIN {X 0.050,Y -228.369,Z 1361.790,A 0.000,B 0.000,C 90.000,E1 322.110} C_DIS
LIN {X -0.027,Y -235.222,Z 1361.773,A 0.000,B 0.000,C 90.000,E1 319.094} C_DIS
LIN {X -0.163,Y -242.834,Z 1361.756,A 0.000,B 0.000,C 90.000,E1 316.134} C_DIS
LIN {X 0.090,Y -252.354,Z 1361.738,A 0.000,B 0.000,C 90.000,E1 312.771} C_DIS
LIN {X 0.057,Y -260.856,Z 1361.724,A 0.000,B 0.000,C 90.000,E1 310.253} C_DIS
LIN {X -0.123,Y -270.355,Z 1361.710,A 0.000,B 0.000,C 90.000,E1 307.810} C_DIS
LIN {X -0.058,Y -280.836,Z 1361.696,A 0.000,B 0.000,C 90.000,E1 305.358} C_DIS
LIN {X 0.046,Y -289.193,Z 1361.687,A 0.000,B 0.000,C 90.000,E1 303.627} C_DIS
LIN {X 0.127,Y -298.455,Z 1361.677,A 0.000,B 0.000,C 90.000,E1 301.926} C_DIS
LIN {X 0.178,Y -306.733,Z 1361.670,A 0.000,B 0.000,C 90.000,E1 300.590} C_DIS
LIN {X -0.092,Y -315.938,Z 1361.663,A 0.000,B 0.000,C 90.000,E1 299.333} C_DIS
LIN {X -0.011,Y -336.505,Z 1361.649,A 0.000,B 0.000,C 90.000,E1 296.796} C_DIS
LIN {X 0.133,Y -349.746,Z 1361.641,A 0.000,B 0.000,C 90.000,E1 295.283} C_DIS
LIN {X 0.127,Y -363.006,Z 1361.632,A 0.000,B 0.000,C 90.000,E1 293.823} C_DIS
LIN {X -0.022,Y -373.373,Z 1361.626,A 0.000,B 0.000,C 90.000,E1 292.695} C_DIS
LIN {X -0.165,Y -385.932,Z 1361.618,A 0.000,B 0.000,C 90.000,E1 291.280} C_DIS
LIN {X 0.118,Y -398.262,Z 1361.610,A 0.000,B 0.000,C 90.000,E1 289.812} C_DIS
LIN {X -0.003,Y -415.414,Z 1361.599,A 0.000,B 0.000,C 90.000,E1 287.873} C_DIS
LIN {X -0.090,Y -424.971,Z 1361.593,A 0.000,B 0.000,C 90.000,E1 286.804} C_DIS
LIN {X 0.080,Y -431.751,Z 1361.589,A 0.000,B 0.000,C 90.000,E1 285.969} C_DIS
LIN {X -0.099,Y -437.887,Z 1361.584,A 0.000,B 0.000,C 90.000,E1 285.190} C_DIS
LIN {X 0.191,Y -443.351,Z 1361.580,A 0.000,B 0.000,C 90.000,E1 284.356} C_DIS
LIN {X -0.003,Y -448.031,Z 1361.576,A 0.000,B 0.000,C 90.000,E1 283.592} C_DIS
LIN {X -0.160,Y -451.905,Z 1361.571,A 0.000,B 0.000,C 90.000,E1 282.827} C_DIS
LIN {X -0.098,Y -454.039,Z 1361.568,A 0.000,B 0.000,C 90.000,E1 282.299} C_DIS
LIN {X -0.020,Y -455.816,Z 1361.565,A 0.000,B 0.000,C 90.000,E1 281.771} C_DIS
LIN {X 0.062,Y -457.270,Z 1361.563,A 0.000,B 0.000,C 90.000,E1 281.243} C_DIS
LIN {X 0.153,Y -458.328,Z 1361.560,A 0.000,B 0.000,C 90.000,E1 280.715} C_DIS
LIN {X 0.170,Y -458.949,Z 1361.557,A 0.000,B 0.000,C 90.000,E1 280.197} C_DIS
LIN {X -0.178,Y -459.092,Z 1361.554,A 0.000,B 0.000,C 90.000,E1 279.726} C_DIS
LIN {X -0.148,Y -458.776,Z 1361.551,A 0.000,B 0.000,C 90.000,E1 279.208} C_DIS
LIN {X -0.043,Y -457.955,Z 1361.548,A 0.000,B 0.000,C 90.000,E1 278.681} C_DIS
LIN {X -0.011,Y -456.635,Z 1361.545,A 0.000,B 0.000,C 90.000,E1 278.163} C_DIS
LIN {X -0.165,Y -453.715,Z 1361.541,A 0.000,B 0.000,C 90.000,E1 277.409} C_DIS
LIN {X -0.151,Y -451.042,Z 1361.538,A 0.000,B 0.000,C 90.000,E1 276.891} C_DIS
LIN {X -0.152,Y -447.764,Z 1361.535,A 0.000,B 0.000,C 90.000,E1 276.372} C_DIS
LIN {X -0.170,Y -443.868,Z 1361.532,A 0.000,B 0.000,C 90.000,E1 275.853} C_DIS
LIN {X 0.229,Y -439.056,Z 1361.530,A 0.000,B 0.000,C 90.000,E1 275.277} C_DIS
LIN {X -0.034,Y -436.254,Z 1361.528,A 0.000,B 0.000,C 90.000,E1 275.049} C_DIS
LIN {X -0.150,Y -433.329,Z 1361.527,A 0.000,B 0.000,C 90.000,E1 274.821} C_DIS
LIN {X -0.059,Y -427.008,Z 1361.524,A 0.000,B 0.000,C 90.000,E1 274.359} C_DIS
LIN {X 0.062,Y -420.602,Z 1361.522,A 0.000,B 0.000,C 90.000,E1 273.955} C_DIS
LIN {X 0.059,Y -414.075,Z 1361.520,A 0.000,B 0.000,C 90.000,E1 273.612} C_DIS
LIN {X -0.096,Y -407.518,Z 1361.518,A 0.000,B 0.000,C 90.000,E1 273.326} C_DIS
LIN {X -0.126,Y -397.209,Z 1361.516,A 0.000,B 0.000,C 90.000,E1 272.922} C_DIS
LIN {X -0.033,Y -387.097,Z 1361.514,A 0.000,B 0.000,C 90.000,E1 272.579} C_DIS
LIN {X -0.127,Y -380.047,Z 1361.513,A 0.000,B 0.000,C 90.000,E1 272.407} C_DIS
LIN {X -0.007,Y -372.107,Z 1361.512,A 0.000,B 0.000,C 90.000,E1 272.236} C_DIS
LIN {X 0.064,Y -355.084,Z 1361.511,A 0.000,B 0.000,C 90.000,E1 272.007} C_DIS
LIN {X -0.131,Y -345.683,Z 1361.511,A 0.000,B 0.000,C 90.000,E1 271.949} C_DIS
LIN {X -0.085,Y -330.573,Z 1361.510,A 0.000,B 0.000,C 90.000,E1 271.892} C_DIS
LIN {X -0.066,Y -181.284,Z 1361.510,A 0.000,B 0.000,C 90.000,E1 271.892} C_DIS
LIN {X -0.072,Y -181.578,Z 1361.501,A 0.000,B 0.000,C 90.000,E1 270.172} C_DIS
LIN {X -0.083,Y -180.881,Z 1361.473,A 0.000,B 0.000,C 90.000,E1 265.122} C_DIS
LIN {X -0.023,Y -179.000,Z 1361.445,A 0.000,B 0.000,C 90.000,E1 260.038} C_DIS
LIN {X 0.071,Y -178.595,Z 1361.440,A 0.000,B 0.000,C 90.000,E1 259.162} C_DIS
LIN {X -0.035,Y -175.648,Z 1361.412,A 0.000,B 0.000,C 90.000,E1 254.102} C_DIS
LIN {X -0.029,Y -172.367,Z 1361.388,A 0.000,B 0.000,C 90.000,E1 249.826} C_DIS
LIN {X -0.016,Y -171.157,Z 1361.378,A 0.000,B 0.000,C 90.000,E1 248.103} C_DIS
LIN {X 0.029,Y -167.457,Z 1361.354,A 0.000,B 0.000,C 90.000,E1 243.768} C_DIS
LIN {X -0.038,Y -166.853,Z 1361.349,A 0.000,B 0.000,C 90.000,E1 242.922} C_DIS
LIN {X 0.027,Y -162.839,Z 1361.325,A 0.000,B 0.000,C 90.000,E1 238.535} C_DIS
LIN {X 0.002,Y -161.522,Z 1361.315,A 0.000,B 0.000,C 90.000,E1 236.786} C_DIS
LIN {X 0.042,Y -157.521,Z 1361.291,A 0.000,B 0.000,C 90.000,E1 232.351} C_DIS
LIN {X -0.025,Y -155.546,Z 1361.276,A 0.000,B 0.000,C 90.000,E1 229.703} C_DIS
LIN {X 0.017,Y -151.839,Z 1361.251,A 0.000,B 0.000,C 90.000,E1 225.202} C_DIS
LIN {X -0.076,Y -150.057,Z 1361.236,A 0.000,B 0.000,C 90.000,E1 222.528} C_DIS
LIN {X -0.041,Y -146.868,Z 1361.211,A 0.000,B 0.000,C 90.000,E1 217.971} C_DIS
LIN {X -0.051,Y -145.453,Z 1361.196,A 0.000,B 0.000,C 90.000,E1 215.231} C_DIS
LIN {X 0.061,Y -142.870,Z 1361.170,A 0.000,B 0.000,C 90.000,E1 210.590} C_DIS
LIN {X -0.012,Y -141.487,Z 1361.150,A 0.000,B 0.000,C 90.000,E1 206.924} C_DIS
LIN {X -0.027,Y -139.384,Z 1361.113,A 0.000,B 0.000,C 90.000,E1 200.429} C_DIS
LIN {X -0.039,Y -138.839,Z 1361.098,A 0.000,B 0.000,C 90.000,E1 197.638} C_DIS
LIN {X 0.022,Y -138.353,Z 1361.056,A 0.000,B 0.000,C 90.000,E1 190.141} C_DIS
LIN {X 0.017,Y -139.522,Z 1361.005,A 0.000,B 0.000,C 90.000,E1 180.802} C_DIS
LIN {X -0.042,Y -141.185,Z 1360.974,A 0.000,B 0.000,C 90.000,E1 175.241} C_DIS
LIN {X 0.070,Y -142.563,Z 1360.958,A 0.000,B 0.000,C 90.000,E1 172.413} C_DIS
LIN {X -0.005,Y -144.847,Z 1360.932,A 0.000,B 0.000,C 90.000,E1 167.825} C_DIS
LIN {X -0.020,Y -147.471,Z 1360.912,A 0.000,B 0.000,C 90.000,E1 164.157} C_DIS
LIN {X 0.007,Y -150.056,Z 1360.892,A 0.000,B 0.000,C 90.000,E1 160.496} C_DIS
LIN {X 0.012,Y -153.400,Z 1360.871,A 0.000,B 0.000,C 90.000,E1 156.869} C_DIS
LIN {X 0.059,Y -155.931,Z 1360.857,A 0.000,B 0.000,C 90.000,E1 154.152} C_DIS
LIN {X 0.032,Y -159.799,Z 1360.837,A 0.000,B 0.000,C 90.000,E1 150.589} C_DIS
LIN {X 0.018,Y -162.039,Z 1360.827,A 0.000,B 0.000,C 90.000,E1 148.820} C_DIS
LIN {X -0.008,Y -166.234,Z 1360.807,A 0.000,B 0.000,C 90.000,E1 145.308} C_DIS
LIN {X -0.007,Y -171.251,Z 1360.788,A 0.000,B 0.000,C 90.000,E1 141.823} C_DIS
LIN {X -0.083,Y -176.140,Z 1360.769,A 0.000,B 0.000,C 90.000,E1 138.405} C_DIS
LIN {X 0.032,Y -180.408,Z 1360.755,A 0.000,B 0.000,C 90.000,E1 135.810} C_DIS
LIN {X 0.008,Y -185.814,Z 1360.736,A 0.000,B 0.000,C 90.000,E1 132.447} C_DIS
LIN {X 0.062,Y -190.434,Z 1360.722,A 0.000,B 0.000,C 90.000,E1 129.930} C_DIS
LIN {X 0.114,Y -197.758,Z 1360.699,A 0.000,B 0.000,C 90.000,E1 125.804} C_DIS
LIN {X 0.027,Y -199.208,Z 1360.695,A 0.000,B 0.000,C 90.000,E1 125.105} C_DIS
LIN {X 0.007,Y -309.517,Z 1360.695,A 0.000,B 0.000,C 90.000,E1 125.105} C_DIS
LIN {X -0.011,Y -312.758,Z 1360.695,A 0.000,B 0.000,C 90.000,E1 125.025} C_DIS
LIN {X 0.090,Y -316.049,Z 1360.693,A 0.000,B 0.000,C 90.000,E1 124.818} C_DIS
LIN {X 0.001,Y -319.660,Z 1360.692,A 0.000,B 0.000,C 90.000,E1 124.485} C_DIS
LIN {X 0.154,Y -323.177,Z 1360.689,A 0.000,B 0.000,C 90.000,E1 123.913} C_DIS
LIN {X -0.035,Y -324.616,Z 1360.687,A 0.000,B 0.000,C 90.000,E1 123.627} C_DIS
LIN {X 0.169,Y -337.426,Z 1360.668,A 0.000,B 0.000,C 90.000,E1 120.129} C_DIS
LIN {X -0.009,Y -349.346,Z 1360.652,A 0.000,B 0.000,C 90.000,E1 117.385} C_DIS
LIN {X 0.140,Y -362.724,Z 1360.637,A 0.000,B 0.000,C 90.000,E1 114.643} C_DIS
LIN {X 0.128,Y -375.930,Z 1360.624,A 0.000,B 0.000,C 90.000,E1 112.280} C_DIS
LIN {X -0.054,Y -390.468,Z 1360.611,A 0.000,B 0.000,C 90.000,E1 109.993} C_DIS
LIN {X 0.220,Y -406.442,Z 1360.599,A 0.000,B 0.000,C 90.000,E1 107.692} C_DIS
LIN {X -0.142,Y -423.961,Z 1360.586,A 0.000,B 0.000,C 90.000,E1 105.536} C_DIS
LIN {X 0.131,Y -443.120,Z 1360.574,A 0.000,B 0.000,C 90.000,E1 103.355} C_DIS
LIN {X 0.021,Y -463.213,Z 1360.563,A 0.000,B 0.000,C 90.000,E1 101.366} C_DIS
LIN {X 0.209,Y -481.195,Z 1360.554,A 0.000,B 0.000,C 90.000,E1 99.726} C_DIS
LIN {X -0.241,Y -483.257,Z 1360.553,A 0.000,B 0.000,C 90.000,E1 99.557} C_DIS
LIN {X 0.119,Y -484.994,Z 1360.552,A 0.000,B 0.000,C 90.000,E1 99.265} C_DIS
LIN {X 0.001,Y -486.294,Z 1360.550,A 0.000,B 0.000,C 90.000,E1 99.029} C_DIS
LIN {X 0.190,Y -487.902,Z 1360.547,A 0.000,B 0.000,C 90.000,E1 98.511} C_DIS
LIN {X -0.093,Y -488.438,Z 1360.545,A 0.000,B 0.000,C 90.000,E1 98.049} C_DIS
LIN {X 0.116,Y -487.991,Z 1360.542,A 0.000,B 0.000,C 90.000,E1 97.530} C_DIS
LIN {X -0.153,Y -486.493,Z 1360.539,A 0.000,B 0.000,C 90.000,E1 97.068} C_DIS
LIN {X 0.223,Y -485.270,Z 1360.538,A 0.000,B 0.000,C 90.000,E1 96.777} C_DIS
LIN {X -0.057,Y -481.785,Z 1360.535,A 0.000,B 0.000,C 90.000,E1 96.315} C_DIS
LIN {X 0.227,Y -469.737,Z 1360.525,A 0.000,B 0.000,C 90.000,E1 94.531} C_DIS
LIN {X -0.014,Y -459.773,Z 1360.517,A 0.000,B 0.000,C 90.000,E1 93.037} C_DIS
LIN {X -0.141,Y -440.285,Z 1360.500,A 0.000,B 0.000,C 90.000,E1 89.943} C_DIS
LIN {X -0.137,Y -428.438,Z 1360.488,A 0.000,B 0.000,C 90.000,E1 87.822} C_DIS
LIN {X -0.072,Y -418.157,Z 1360.477,A 0.000,B 0.000,C 90.000,E1 85.927} C_DIS
LIN {X -0.223,Y -407.754,Z 1360.467,A 0.000,B 0.000,C 90.000,E1 84.033} C_DIS
LIN {X -0.140,Y -398.693,Z 1360.457,A 0.000,B 0.000,C 90.000,E1 82.356} C_DIS
LIN {X 0.167,Y -389.414,Z 1360.448,A 0.000,B 0.000,C 90.000,E1 80.622} C_DIS
LIN {X 0.048,Y -379.949,Z 1360.438,A 0.000,B 0.000,C 90.000,E1 78.926} C_DIS
LIN {X 0.138,Y -370.327,Z 1360.429,A 0.000,B 0.000,C 90.000,E1 77.173} C_DIS
LIN {X 0.126,Y -360.477,Z 1360.419,A 0.000,B 0.000,C 90.000,E1 75.408} C_DIS
LIN {X 0.121,Y -350.581,Z 1360.409,A 0.000,B 0.000,C 90.000,E1 73.614} C_DIS
LIN {X -0.056,Y -340.552,Z 1360.399,A 0.000,B 0.000,C 90.000,E1 71.819} C_DIS
LIN {X -0.020,Y -328.904,Z 1360.387,A 0.000,B 0.000,C 90.000,E1 69.645} C_DIS
LIN {X -0.083,Y -312.813,Z 1360.369,A 0.000,B 0.000,C 90.000,E1 66.485} C_DIS
LIN {X -0.141,Y -301.021,Z 1360.355,A 0.000,B 0.000,C 90.000,E1 63.896} C_DIS
LIN {X 0.032,Y -289.317,Z 1360.338,A 0.000,B 0.000,C 90.000,E1 60.873} C_DIS
LIN {X -0.091,Y -282.358,Z 1360.327,A 0.000,B 0.000,C 90.000,E1 58.869} C_DIS
LIN {X 0.143,Y -272.078,Z 1360.308,A 0.000,B 0.000,C 90.000,E1 55.388} C_DIS
LIN {X -0.054,Y -264.362,Z 1360.292,A 0.000,B 0.000,C 90.000,E1 52.637} C_DIS
LIN {X -0.078,Y -255.128,Z 1360.273,A 0.000,B 0.000,C 90.000,E1 49.094} C_DIS
LIN {X -0.096,Y -246.423,Z 1360.253,A 0.000,B 0.000,C 90.000,E1 45.486} C_DIS
LIN {X 0.132,Y -238.523,Z 1360.232,A 0.000,B 0.000,C 90.000,E1 41.757} C_DIS
LIN {X 0.021,Y -231.446,Z 1360.211,A 0.000,B 0.000,C 90.000,E1 38.051} C_DIS
LIN {X -0.032,Y -225.226,Z 1360.190,A 0.000,B 0.000,C 90.000,E1 34.278} C_DIS
LIN {X -0.100,Y -219.950,Z 1360.169,A 0.000,B 0.000,C 90.000,E1 30.463} C_DIS
LIN {X -0.051,Y -214.969,Z 1360.143,A 0.000,B 0.000,C 90.000,E1 25.796} C_DIS
LIN {X -0.063,Y -211.350,Z 1360.117,A 0.000,B 0.000,C 90.000,E1 21.099} C_DIS
LIN {X -0.036,Y -208.950,Z 1360.095,A 0.000,B 0.000,C 90.000,E1 17.149} C_DIS
LIN {X 0.062,Y -207.137,Z 1360.078,A 0.000,B 0.000,C 90.000,E1 13.953} C_DIS
LIN {X 0.025,Y -205.511,Z 1360.060,A 0.000,B 0.000,C 90.000,E1 10.782} C_DIS
LIN {X 0.069,Y -203.597,Z 1360.038,A 0.000,B 0.000,C 90.000,E1 6.777} C_DIS
LIN {X -0.076,Y -202.271,Z 1360.020,A 0.000,B 0.000,C 90.000,E1 3.612} C_DIS
LIN {X -0.049,Y -200.776,Z 1359.993,A 0.000,B 0.000,C 90.000,E1 358.740} C_DIS
LIN {X -0.104,Y -200.183,Z 1359.962,A 0.000,B 0.000,C 90.000,E1 353.109} C_DIS
LIN {X 0.080,Y -201.806,Z 1359.917,A 0.000,B 0.000,C 90.000,E1 344.991} C_DIS
LIN {X 0.012,Y -204.971,Z 1359.885,A 0.000,B 0.000,C 90.000,E1 339.390} C_DIS
LIN {X 0.084,Y -209.193,Z 1359.859,A 0.000,B 0.000,C 90.000,E1 334.588} C_DIS
LIN {X -0.021,Y -213.928,Z 1359.837,A 0.000,B 0.000,C 90.000,E1 330.667} C_DIS
LIN {X -0.005,Y -219.904,Z 1359.815,A 0.000,B 0.000,C 90.000,E1 326.755} C_DIS
LIN {X -0.107,Y -226.976,Z 1359.794,A 0.000,B 0.000,C 90.000,E1 322.924} C_DIS
LIN {X 0.104,Y -233.580,Z 1359.777,A 0.000,B 0.000,C 90.000,E1 319.828} C_DIS
LIN {X -0.050,Y -240.990,Z 1359.760,A 0.000,B 0.000,C 90.000,E1 316.863} C_DIS
LIN {X -0.039,Y -250.239,Z 1359.742,A 0.000,B 0.000,C 90.000,E1 313.542} C_DIS
LIN {X 0.043,Y -258.434,Z 1359.728,A 0.000,B 0.000,C 90.000,E1 310.987} C_DIS
LIN {X -0.027,Y -267.641,Z 1359.714,A 0.000,B 0.000,C 90.000,E1 308.508} C_DIS
LIN {X -0.087,Y -279.389,Z 1359.698,A 0.000,B 0.000,C 90.000,E1 305.724} C_DIS
LIN {X -0.009,Y -287.562,Z 1359.689,A 0.000,B 0.000,C 90.000,E1 303.992} C_DIS
LIN {X 0.053,Y -296.645,Z 1359.679,A 0.000,B 0.000,C 90.000,E1 302.291} C_DIS
LIN {X -0.177,Y -304.695,Z 1359.672,A 0.000,B 0.000,C 90.000,E1 301.003} C_DIS
LIN {X -0.050,Y -313.636,Z 1359.665,A 0.000,B 0.000,C 90.000,E1 299.667} C_DIS
LIN {X 0.070,Y -323.528,Z 1359.658,A 0.000,B 0.000,C 90.000,E1 298.359} C_DIS
LIN {X 0.089,Y -347.190,Z 1359.642,A 0.000,B 0.000,C 90.000,E1 295.591} C_DIS
LIN {X 0.013,Y -360.513,Z 1359.634,A 0.000,B 0.000,C 90.000,E1 294.131} C_DIS
LIN {X 0.152,Y -370.964,Z 1359.628,A 0.000,B 0.000,C 90.000,E1 292.950} C_DIS
LIN {X -0.012,Y -383.580,Z 1359.620,A 0.000,B 0.000,C 90.000,E1 291.535} C_DIS
LIN {X -0.142,Y -395.986,Z 1359.612,A 0.000,B 0.000,C 90.000,E1 290.120} C_DIS
LIN {X -0.021,Y -410.701,Z 1359.602,A 0.000,B 0.000,C 90.000,E1 288.417} C_DIS
LIN {X -0.018,Y -422.891,Z 1359.595,A 0.000,B 0.000,C 90.000,E1 287.040} C_DIS
LIN {X 0.139,Y -429.779,Z 1359.590,A 0.000,B 0.000,C 90.000,E1 286.205} C_DIS
LIN {X -0.063,Y -436.166,Z 1359.586,A 0.000,B 0.000,C 90.000,E1 285.426} C_DIS
LIN {X 0.217,Y -441.836,Z 1359.581,A 0.000,B 0.000,C 90.000,E1 284.592} C_DIS
LIN {X 0.217,Y -445.247,Z 1359.578,A 0.000,B 0.000,C 90.000,E1 284.064} C_DIS
LIN {X 0.036,Y -449.654,Z 1359.574,A 0.000,B 0.000,C 90.000,E1 283.300} C_DIS
LIN {X 0.086,Y -452.160,Z 1359.571,A 0.000,B 0.000,C 90.000,E1 282.771} C_DIS
LIN {X 0.153,Y -454.273,Z 1359.568,A 0.000,B 0.000,C 90.000,E1 282.243} C_DIS
LIN {X -0.213,Y -456.090,Z 1359.565,A 0.000,B 0.000,C 90.000,E1 281.771} C_DIS
LIN {X -0.130,Y -457.521,Z 1359.562,A 0.000,B 0.000,C 90.000,E1 281.243} C_DIS
LIN {X -0.038,Y -458.607,Z 1359.559,A 0.000,B 0.000,C 90.000,E1 280.715} C_DIS
LIN {X -0.020,Y -459.192,Z 1359.557,A 0.000,B 0.000,C 90.000,E1 280.197} C_DIS
LIN {X 0.086,Y -459.354,Z 1359.554,A 0.000,B 0.000,C 90.000,E1 279.670} C_DIS
LIN {X 0.119,Y -459.050,Z 1359.551,A 0.000,B 0.000,C 90.000,E1 279.151} C_DIS
LIN {X 0.224,Y -458.250,Z 1359.548,A 0.000,B 0.000,C 90.000,E1 278.624} C_DIS
LIN {X -0.194,Y -456.967,Z 1359.545,A 0.000,B 0.000,C 90.000,E1 278.163} C_DIS
LIN {X 0.105,Y -453.996,Z 1359.541,A 0.000,B 0.000,C 90.000,E1 277.352} C_DIS
LIN {X 0.120,Y -451.303,Z 1359.538,A 0.000,B 0.000,C 90.000,E1 276.834} C_DIS
LIN {X 0.120,Y -448.059,Z 1359.535,A 0.000,B 0.000,C 90.000,E1 276.315} C_DIS
LIN {X 0.102,Y -444.154,Z 1359.532,A 0.000,B 0.000,C 90.000,E1 275.796} C_DIS
LIN {X 0.063,Y -439.358,Z 1359.529,A 0.000,B 0.000,C 90.000,E1 275.277} C_DIS
LIN {X -0.199,Y -436.596,Z 1359.528,A 0.000,B 0.000,C 90.000,E1 275.049} C_DIS
LIN {X 0.004,Y -430.355,Z 1359.525,A 0.000,B 0.000,C 90.000,E1 274.531} C_DIS
LIN {X -0.145,Y -423.996,Z 1359.523,A 0.000,B 0.000,C 90.000,E1 274.131} C_DIS
LIN {X 0.112,Y -417.421,Z 1359.521,A 0.000,B 0.000,C 90.000,E1 273.726} C_DIS
LIN {X 0.030,Y -407.739,Z 1359.518,A 0.000,B 0.000,C 90.000,E1 273.269} C_DIS
LIN {X 0.110,Y -401.000,Z 1359.517,A 0.000,B 0.000,C 90.000,E1 272.980} C_DIS
LIN {X 0.008,Y -394.136,Z 1359.515,A 0.000,B 0.000,C 90.000,E1 272.751} C_DIS
LIN {X 0.124,Y -387.399,Z 1359.514,A 0.000,B 0.000,C 90.000,E1 272.522} C_DIS
LIN {X 0.047,Y -380.321,Z 1359.513,A 0.000,B 0.000,C 90.000,E1 272.350} C_DIS
LIN {X 0.168,Y -372.474,Z 1359.512,A 0.000,B 0.000,C 90.000,E1 272.178} C_DIS
LIN {X 0.123,Y -363.639,Z 1359.512,A 0.000,B 0.000,C 90.000,E1 272.064} C_DIS
LIN {X -0.026,Y -351.351,Z 1359.511,A 0.000,B 0.000,C 90.000,E1 271.949} C_DIS
LIN {X -0.140,Y -337.775,Z 1359.510,A 0.000,B 0.000,C 90.000,E1 271.892} C_DIS
LIN {X 0.072,Y -181.285,Z 1359.510,A 0.000,B 0.000,C 90.000,E1 271.835} C_DIS
LIN {X -0.035,Y -181.580,Z 1359.502,A 0.000,B 0.000,C 90.000,E1 270.344} C_DIS
LIN {X -0.017,Y -180.795,Z 1359.471,A 0.000,B 0.000,C 90.000,E1 264.780} C_DIS
LIN {X 0.056,Y -178.895,Z 1359.443,A 0.000,B 0.000,C 90.000,E1 259.690} C_DIS
LIN {X -0.038,Y -175.938,Z 1359.415,A 0.000,B 0.000,C 90.000,E1 254.629} C_DIS
LIN {X 0.077,Y -175.390,Z 1359.410,A 0.000,B 0.000,C 90.000,E1 253.740} C_DIS
LIN {X -0.087,Y -172.161,Z 1359.386,A 0.000,B 0.000,C 90.000,E1 249.518} C_DIS
LIN {X -0.048,Y -171.629,Z 1359.381,A 0.000,B 0.000,C 90.000,E1 248.646} C_DIS
LIN {X -0.053,Y -167.851,Z 1359.357,A 0.000,B 0.000,C 90.000,E1 244.332} C_DIS
LIN {X 0.039,Y -166.582,Z 1359.348,A 0.000,B 0.000,C 90.000,E1 242.564} C_DIS
LIN {X 0.025,Y -162.573,Z 1359.323,A 0.000,B 0.000,C 90.000,E1 238.201} C_DIS
LIN {X 0.084,Y -161.255,Z 1359.314,A 0.000,B 0.000,C 90.000,E1 236.421} C_DIS
LIN {X -0.006,Y -157.257,Z 1359.289,A 0.000,B 0.000,C 90.000,E1 232.029} C_DIS
LIN {X -0.079,Y -155.979,Z 1359.279,A 0.000,B 0.000,C 90.000,E1 230.275} C_DIS
LIN {X 0.097,Y -152.234,Z 1359.254,A 0.000,B 0.000,C 90.000,E1 225.729} C_DIS
LIN {X 0.008,Y -150.475,Z 1359.239,A 0.000,B 0.000,C 90.000,E1 223.056} C_DIS
LIN {X -0.063,Y -147.200,Z 1359.214,A 0.000,B 0.000,C 90.000,E1 218.543} C_DIS
LIN {X -0.010,Y -145.220,Z 1359.194,A 0.000,B 0.000,C 90.000,E1 214.865} C_DIS
LIN {X 0.018,Y -142.349,Z 1359.163,A 0.000,B 0.000,C 90.000,E1 209.333} C_DIS
LIN {X -0.054,Y -141.736,Z 1359.153,A 0.000,B 0.000,C 90.000,E1 207.513} C_DIS
LIN {X 0.053,Y -139.486,Z 1359.117,A 0.000,B 0.000,C 90.000,E1 200.972} C_DIS
LIN {X 0.042,Y -138.987,Z 1359.101,A 0.000,B 0.000,C 90.000,E1 198.181} C_DIS
LIN {X 0.003,Y -138.334,Z 1359.054,A 0.000,B 0.000,C 90.000,E1 189.792} C_DIS
LIN {X 0.027,Y -139.423,Z 1359.008,A 0.000,B 0.000,C 90.000,E1 181.375} C_DIS
LIN {X -0.059,Y -141.343,Z 1358.972,A 0.000,B 0.000,C 90.000,E1 174.894} C_DIS
LIN {X 0.058,Y -142.698,Z 1358.956,A 0.000,B 0.000,C 90.000,E1 172.064} C_DIS
LIN {X 0.017,Y -145.067,Z 1358.930,A 0.000,B 0.000,C 90.000,E1 167.465} C_DIS
LIN {X 0.014,Y -147.692,Z 1358.910,A 0.000,B 0.000,C 90.000,E1 163.795} C_DIS
LIN {X 0.047,Y -150.341,Z 1358.890,A 0.000,B 0.000,C 90.000,E1 160.134} C_DIS
LIN {X 0.041,Y -154.595,Z 1358.865,A 0.000,B 0.000,C 90.000,E1 155.613} C_DIS
LIN {X 0.049,Y -158.134,Z 1358.845,A 0.000,B 0.000,C 90.000,E1 152.025} C_DIS
LIN {X 0.008,Y -162.421,Z 1358.825,A 0.000,B 0.000,C 90.000,E1 148.486} C_DIS
LIN {X -0.010,Y -166.678,Z 1358.805,A 0.000,B 0.000,C 90.000,E1 144.975} C_DIS
LIN {X -0.003,Y -171.683,Z 1358.786,A 0.000,B 0.000,C 90.000,E1 141.492} C_DIS
LIN {X -0.094,Y -176.653,Z 1358.767,A 0.000,B 0.000,C 90.000,E1 138.081} C_DIS
LIN {X 0.034,Y -180.950,Z 1358.753,A 0.000,B 0.000,C 90.000,E1 135.486} C_DIS
LIN {X 0.021,Y -186.372,Z 1358.734,A 0.000,B 0.000,C 90.000,E1 132.123} C_DIS
LIN {X -0.038,Y -191.002,Z 1358.720,A 0.000,B 0.000,C 90.000,E1 129.644} C_DIS
LIN {X -0.120,Y -196.780,Z 1358.702,A 0.000,B 0.000,C 90.000,E1 126.377} C_DIS
LIN {X 0.055,Y -199.192,Z 1358.695,A 0.000,B 0.000,C 90.000,E1 125.105} C_DIS
LIN {X 0.051,Y -308.569,Z 1358.695,A 0.000,B 0.000,C 90.000,E1 125.105} C_DIS
LIN {X -0.017,Y -309.990,Z 1358.695,A 0.000,B 0.000,C 90.000,E1 125.105} C_DIS
LIN {X 0.050,Y -314.999,Z 1358.694,A 0.000,B 0.000,C 90.000,E1 124.898} C_DIS
LIN {X 0.118,Y -317.512,Z 1358.693,A 0.000,B 0.000,C 90.000,E1 124.692} C_DIS
LIN {X 0.065,Y -321.322,Z 1358.690,A 0.000,B 0.000,C 90.000,E1 124.246} C_DIS
LIN {X 0.152,Y -323.162,Z 1358.689,A 0.000,B 0.000,C 90.000,E1 123.913} C_DIS
LIN {X -0.029,Y -324.593,Z 1358.687,A 0.000,B 0.000,C 90.000,E1 123.627} C_DIS
LIN {X 0.186,Y -337.394,Z 1358.668,A 0.000,B 0.000,C 90.000,E1 120.129} C_DIS
LIN {X 0.003,Y -349.315,Z 1358.652,A 0.000,B 0.000,C 90.000,E1 117.385} C_DIS
LIN {X 0.155,Y -362.687,Z 1358.637,A 0.000,B 0.000,C 90.000,E1 114.643} C_DIS
LIN {X 0.143,Y -375.892,Z 1358.624,A 0.000,B 0.000,C 90.000,E1 112.280} C_DIS
LIN {X -0.038,Y -390.429,Z 1358.611,A 0.000,B 0.000,C 90.000,E1 109.993} C_DIS
LIN {X 0.235,Y -406.399,Z 1358.599,A 0.000,B 0.000,C 90.000,E1 107.692} C_DIS
